LIN {X 0,Y 426.139,Z 463.604,A -85,B 0,C 180,E1 -9930.748,E2 -9930.748} C_VEL
LIN {X 0,Y 426.519,Z 456.049,A -85,B 0,C 180,E1 -9931.425,E2 -9931.425} C_VEL
LIN {X 0,Y 426.812,Z 447.127,A -85,B 0,C 180,E1 -9932.076,E2 -9932.076} C_VEL
LIN {X 0,Y 427.163,Z 437.86,A -85,B 0,C 180,E1 -9932.604,E2 -9932.604} C_VEL
LIN {X 0,Y 427.406,Z 427.667,A -85,B 0,C 180,E1 -9933.038,E2 -9933.038} C_VEL
LIN {X 0,Y 427.627,Z 415.432,A -85,B 0,C 180,E1 -9933.376,E2 -9933.376} C_VEL
LIN {X 0,Y 428.378,Z 356.063,A -85,B 0,C 180,E1 -9934.529,E2 -9934.529} C_VEL
LIN {X 0,Y 425.875,Z 339.164,A -85,B 0,C 180,E1 -9934.972,E2 -9934.972} C_VEL
LIN {X 0,Y 426.543,Z 323.121,A -85,B 0,C 180,E1 -9938.192,E2 -9938.192} C_VEL
LIN {X 0,Y 427.303,Z 307.169,A -85,B 0,C 180,E1 -9941.454,E2 -9941.454} C_VEL
LIN {X 0,Y 427.541,Z 299.568,A -85,B 0,C 180,E1 -9943.038,E2 -9943.038} C_VEL
LIN {X 0,Y 425.324,Z 287.505,A -85,B 0,C 180,E1 -9945.749,E2 -9945.749} C_VEL
LIN {X 0,Y 425.264,Z 287.509,A -85,B 0,C 180,E1 -9948.623,E2 -9948.623} C_VEL
LIN {X 0,Y 425.272,Z 287.509,A -85,B 0,C 180,E1 -9951.101,E2 -9951.101} C_VEL
LIN {X 0,Y 425.29,Z 287.504,A -85,B 0,C 180,E1 -9954.665,E2 -9954.665} C_VEL
LIN {X 0,Y 425.26,Z 287.513,A -85,B 0,C 180,E1 -9958.074,E2 -9958.074} C_VEL
LIN {X 0,Y 425.296,Z 287.504,A -85,B 0,C 180,E1 -9961.366,E2 -9961.366} C_VEL
LIN {X 0,Y 425.26,Z 287.512,A -85,B 0,C 180,E1 -9964.553,E2 -9964.553} C_VEL
LIN {X 0,Y 425.293,Z 287.504,A -85,B 0,C 180,E1 -9967.731,E2 -9967.731} C_VEL
LIN {X 0,Y 425.333,Z 287.501,A -85,B 0,C 180,E1 -9971.096,E2 -9971.096} C_VEL
LIN {X 0,Y 424.637,Z 287.586,A -85,B 0,C 180,E1 -9971.886,E2 -9971.886} C_VEL
LIN {X 0,Y 421.762,Z 287.946,A -85,B 0,C 180,E1 -9973.17,E2 -9973.17} C_VEL
LIN {X 0,Y 419.363,Z 288.243,A -85,B 0,C 180,E1 -9974.207,E2 -9974.207} C_VEL
LIN {X 0,Y 418.359,Z 288.374,A -85,B 0,C 180,E1 -9975.008,E2 -9975.008} C_VEL
LIN {X 0,Y 418.29,Z 288.377,A -85,B 0,C 180,E1 -9975.279,E2 -9975.279} C_VEL
LIN {X 0,Y 418.316,Z 288.373,A -85,B 0,C 180,E1 -9978.368,E2 -9978.368} C_VEL
LIN {X 0,Y 418.451,Z 288.355,A -85,B 0,C 180,E1 -9982.277,E2 -9982.277} C_VEL
LIN {X 0,Y 418.474,Z 288.353,A -85,B 0,C 180,E1 -9984.215,E2 -9984.215} C_VEL
LIN {X 0,Y 418.536,Z 288.348,A -85,B 0,C 180,E1 -9988.074,E2 -9988.074} C_VEL
LIN {X 0,Y 418.409,Z 288.361,A -85,B 0,C 180,E1 -9990.96,E2 -9990.96} C_VEL
LIN {X 0,Y 418.47,Z 288.353,A -85,B 0,C 180,E1 -9992.886,E2 -9992.886} C_VEL
LIN {X 0,Y 418.471,Z 288.358,A -85,B 0,C 180,E1 -9995.781,E2 -9995.781} C_VEL
LIN {X 0,Y 418.369,Z 288.368,A -85,B 0,C 180,E1 -9998.693,E2 -9998.693} C_VEL
LIN {X 0,Y 418.31,Z 288.374,A -85,B 0,C 180,E1 -10001.628,E2 -10001.628} C_VEL
LIN {X 0,Y 418.297,Z 288.383,A -85,B 0,C 180,E1 -10004.594,E2 -10004.594} C_VEL
LIN {X 0,Y 418.275,Z 288.378,A -85,B 0,C 180,E1 -10007.6,E2 -10007.6} C_VEL
LIN {X 0,Y 418.243,Z 288.386,A -85,B 0,C 180,E1 -10010.659,E2 -10010.659} C_VEL
LIN {X 0,Y 418.263,Z 288.38,A -85,B 0,C 180,E1 -10013.778,E2 -10013.778} C_VEL
LIN {X 0,Y 418.212,Z 288.39,A -85,B 0,C 180,E1 -10017.043,E2 -10017.043} C_VEL
LIN {X 0,Y 418.227,Z 288.384,A -85,B 0,C 180,E1 -10020.268,E2 -10020.268} C_VEL
LIN {X 0,Y 418.23,Z 288.392,A -85,B 0,C 180,E1 -10023.673,E2 -10023.673} C_VEL
LIN {X 0,Y 418.217,Z 288.386,A -85,B 0,C 180,E1 -10027.22,E2 -10027.22} C_VEL
LIN {X 0,Y 418.219,Z 288.388,A -85,B 0,C 180,E1 -10029.678,E2 -10029.678} C_VEL
LIN {X 0,Y 418.201,Z 288.393,A -85,B 0,C 180,E1 -10032.316,E2 -10032.316} C_VEL
LIN {X 0,Y 418.206,Z 288.386,A -85,B 0,C 180,E1 -10035.104,E2 -10035.104} C_VEL
LIN {X 0,Y 418.208,Z 288.387,A -85,B 0,C 180,E1 -10037.762,E2 -10037.762} C_VEL
LIN {X 0,Y 418.218,Z 288.393,A -85,B 0,C 180,E1 -10040.615,E2 -10040.615} C_VEL
LIN {X 0,Y 418.204,Z 288.386,A -85,B 0,C 180,E1 -10043.971,E2 -10043.971} C_VEL
LIN {X 0,Y 418.201,Z 288.389,A -85,B 0,C 180,E1 -10047.467,E2 -10047.467} C_VEL
LIN {X 0,Y 418.233,Z 288.387,A -85,B 0,C 180,E1 -10050.89,E2 -10050.89} C_VEL
LIN {X 0,Y 418.224,Z 288.385,A -85,B 0,C 180,E1 -10054.092,E2 -10054.092} C_VEL
LIN {X 0,Y 418.185,Z 288.393,A -85,B 0,C 180,E1 -10057.26,E2 -10057.26} C_VEL
LIN {X 0,Y 418.232,Z 288.384,A -85,B 0,C 180,E1 -10060.361,E2 -10060.361} C_VEL
LIN {X 0,Y 418.264,Z 288.381,A -85,B 0,C 180,E1 -10063.402,E2 -10063.402} C_VEL
LIN {X 0,Y 418.302,Z 288.374,A -85,B 0,C 180,E1 -10066.992,E2 -10066.992} C_VEL
LIN {X 0,Y 418.303,Z 288.383,A -85,B 0,C 180,E1 -10070.327,E2 -10070.327} C_VEL
LIN {X 0,Y 418.439,Z 288.358,A -85,B 0,C 180,E1 -10073.248,E2 -10073.248} C_VEL
LIN {X 0,Y 418.29,Z 288.377,A -85,B 0,C 180,E1 -10075.18,E2 -10075.18} C_VEL
LIN {X 0,Y 418.489,Z 288.352,A -85,B 0,C 180,E1 -10078.075,E2 -10078.075} C_VEL
LIN {X 0,Y 418.614,Z 288.335,A -85,B 0,C 180,E1 -10079.999,E2 -10079.999} C_VEL
LIN {X 0,Y 418.46,Z 288.36,A -85,B 0,C 180,E1 -10082.888,E2 -10082.888} C_VEL
LIN {X 0,Y 418.437,Z 288.359,A -85,B 0,C 180,E1 -10086.751,E2 -10086.751} C_VEL
LIN {X 0,Y 418.286,Z 288.381,A -85,B 0,C 180,E1 -10089.672,E2 -10089.672} C_VEL
LIN {X 0,Y 418.301,Z 288.375,A -85,B 0,C 180,E1 -10093.007,E2 -10093.007} C_VEL
LIN {X 0,Y 418.258,Z 288.38,A -85,B 0,C 180,E1 -10096.736,E2 -10096.736} C_VEL
LIN {X 0,Y 418.22,Z 288.39,A -85,B 0,C 180,E1 -10099.792,E2 -10099.792} C_VEL
LIN {X 0,Y 418.189,Z 288.39,A -85,B 0,C 180,E1 -10102.738,E2 -10102.738} C_VEL
LIN {X 0,Y 418.221,Z 288.387,A -85,B 0,C 180,E1 -10105.907,E2 -10105.907} C_VEL
LIN {X 0,Y 418.218,Z 288.386,A -85,B 0,C 180,E1 -10109.165,E2 -10109.165} C_VEL
LIN {X 0,Y 418.212,Z 288.393,A -85,B 0,C 180,E1 -10112.847,E2 -10112.847} C_VEL
LIN {X 0,Y 418.203,Z 288.387,A -85,B 0,C 180,E1 -10116.241,E2 -10116.241} C_VEL
LIN {X 0,Y 418.204,Z 288.388,A -85,B 0,C 180,E1 -10119.687,E2 -10119.687} C_VEL
LIN {X 0,Y 418.186,Z 288.389,A -85,B 0,C 180,E1 -10122.324,E2 -10122.324} C_VEL
LIN {X 0,Y 418.2,Z 288.39,A -85,B 0,C 180,E1 -10125.112,E2 -10125.112} C_VEL
LIN {X 0,Y 418.207,Z 288.393,A -85,B 0,C 180,E1 -10127.771,E2 -10127.771} C_VEL
LIN {X 0,Y 418.207,Z 288.39,A -85,B 0,C 180,E1 -10131.56,E2 -10131.56} C_VEL
LIN {X 0,Y 418.224,Z 288.384,A -85,B 0,C 180,E1 -10135.162,E2 -10135.162} C_VEL
LIN {X 0,Y 418.219,Z 288.385,A -85,B 0,C 180,E1 -10137.476,E2 -10137.476} C_VEL
LIN {X 0,Y 418.239,Z 288.388,A -85,B 0,C 180,E1 -10140.902,E2 -10140.902} C_VEL
LIN {X 0,Y 418.255,Z 288.523,A -85,B 0,C 180,E1 -10142.033,E2 -10142.033} C_VEL
LIN {X 0,Y 421.967,Z 305.233,A -85,B 0,C 180,E1 -10145.136,E2 -10145.136} C_VEL
LIN {X 0,Y 422.416,Z 308.453,A -85,B 0,C 180,E1 -10145.706,E2 -10145.706} C_VEL
LIN {X 0,Y 421.093,Z 327.942,A -85,B 0,C 180,E1 -10148.918,E2 -10148.918} C_VEL
LIN {X 0,Y 420.029,Z 345.035,A -85,B 0,C 180,E1 -10151.662,E2 -10151.662} C_VEL
LIN {X 0,Y 422.513,Z 365.547,A -85,B 0,C 180,E1 -10152.142,E2 -10152.142} C_VEL
LIN {X 0,Y 421.378,Z 450.417,A -85,B 0,C 180,E1 -10153.719,E2 -10153.719} C_VEL
LIN {X 0,Y 421.099,Z 459.636,A -85,B 0,C 180,E1 -10153.988,E2 -10153.988} C_VEL
LIN {X 0,Y 420.726,Z 469.267,A -85,B 0,C 180,E1 -10154.377,E2 -10154.377} C_VEL
LIN {X 0,Y 420.344,Z 478.447,A -85,B 0,C 180,E1 -10154.86,E2 -10154.86} C_VEL
LIN {X 0,Y 419.758,Z 489.136,A -85,B 0,C 180,E1 -10155.582,E2 -10155.582} C_VEL
LIN {X 0,Y 419.287,Z 499.136,A -85,B 0,C 180,E1 -10156.432,E2 -10156.432} C_VEL
LIN {X 0,Y 418.893,Z 506.591,A -85,B 0,C 180,E1 -10157.182,E2 -10157.182} C_VEL
LIN {X 0,Y 418.352,Z 516.259,A -85,B 0,C 180,E1 -10158.373,E2 -10158.373} C_VEL
LIN {X 0,Y 417.931,Z 522.899,A -85,B 0,C 180,E1 -10159.343,E2 -10159.343} C_VEL
LIN {X 0,Y 417.616,Z 529.845,A -85,B 0,C 180,E1 -10160.559,E2 -10160.559} C_VEL
LIN {X 0,Y 417.407,Z 535.619,A -85,B 0,C 180,E1 -10161.775,E2 -10161.775} C_VEL
LIN {X 0,Y 417.222,Z 541.176,A -85,B 0,C 180,E1 -10163.231,E2 -10163.231} C_VEL
LIN {X 0,Y 417.147,Z 545.5,A -85,B 0,C 180,E1 -10164.686,E2 -10164.686} C_VEL
LIN {X 0,Y 417.054,Z 548.703,A -85,B 0,C 180,E1 -10166.137,E2 -10166.137} C_VEL
LIN {X 0,Y 417.152,Z 550.338,A -85,B 0,C 180,E1 -10167.105,E2 -10167.105} C_VEL
LIN {X 0,Y 417.104,Z 552.078,A -85,B 0,C 180,E1 -10169.037,E2 -10169.037} C_VEL
LIN {X 0,Y 417.117,Z 552.372,A -85,B 0,C 180,E1 -10170.002,E2 -10170.002} C_VEL
LIN {X 0,Y 417.118,Z 551.594,A -85,B 0,C 180,E1 -10171.933,E2 -10171.933} C_VEL
LIN {X 0,Y 417.122,Z 550.564,A -85,B 0,C 180,E1 -10172.899,E2 -10172.899} C_VEL
LIN {X 0,Y 417.146,Z 547.23,A -85,B 0,C 180,E1 -10174.834,E2 -10174.834} C_VEL
LIN {X 0,Y 417.139,Z 543.557,A -85,B 0,C 180,E1 -10176.264,E2 -10176.264} C_VEL
LIN {X 0,Y 417.301,Z 538.557,A -85,B 0,C 180,E1 -10177.744,E2 -10177.744} C_VEL
LIN {X 0,Y 417.555,Z 532.315,A -85,B 0,C 180,E1 -10179.202,E2 -10179.202} C_VEL
LIN {X 0,Y 417.871,Z 525.97,A -85,B 0,C 180,E1 -10180.417,E2 -10180.417} C_VEL
LIN {X 0,Y 418.36,Z 518.307,A -85,B 0,C 180,E1 -10181.631,E2 -10181.631} C_VEL
LIN {X 0,Y 418.762,Z 511.042,A -85,B 0,C 180,E1 -10182.603,E2 -10182.603} C_VEL
LIN {X 0,Y 419.366,Z 502.16,A -85,B 0,C 180,E1 -10183.592,E2 -10183.592} C_VEL
LIN {X 0,Y 419.968,Z 493.44,A -85,B 0,C 180,E1 -10184.402,E2 -10184.402} C_VEL
LIN {X 0,Y 420.56,Z 483.816,A -85,B 0,C 180,E1 -10185.136,E2 -10185.136} C_VEL
LIN {X 0,Y 421.18,Z 472.887,A -85,B 0,C 180,E1 -10185.795,E2 -10185.795} C_VEL
LIN {X 0,Y 421.67,Z 462.526,A -85,B 0,C 180,E1 -10186.273,E2 -10186.273} C_VEL
LIN {X 0,Y 422.057,Z 451.679,A -85,B 0,C 180,E1 -10186.631,E2 -10186.631} C_VEL
LIN {X 0,Y 422.44,Z 432.575,A -85,B 0,C 180,E1 -10187.02,E2 -10187.02} C_VEL
LIN {X 0,Y 423.325,Z 363.978,A -85,B 0,C 180,E1 -10188.327,E2 -10188.327} C_VEL
LIN {X 0,Y 420.546,Z 343.811,A -85,B 0,C 180,E1 -10188.906,E2 -10188.906} C_VEL
LIN {X 0,Y 421.697,Z 323.527,A -85,B 0,C 180,E1 -10192.023,E2 -10192.023} C_VEL
LIN {X 0,Y 422.6,Z 308.661,A -85,B 0,C 180,E1 -10194.313,E2 -10194.313} C_VEL
LIN {X 0,Y 421.537,Z 301.939,A -85,B 0,C 180,E1 -10195.465,E2 -10195.465} C_VEL
LIN {X 0,Y 418.732,Z 290.403,A -85,B 0,C 180,E1 -10197.546,E2 -10197.546} C_VEL
LIN {X 0,Y 418.215,Z 288.398,A -85,B 0,C 180,E1 -10197.947,E2 -10197.947} C_VEL
LIN {X 0,Y 418.232,Z 288.393,A -85,B 0,C 180,E1 -10201.019,E2 -10201.019} C_VEL
LIN {X 0,Y 418.24,Z 288.389,A -85,B 0,C 180,E1 -10203.676,E2 -10203.676} C_VEL
LIN {X 0,Y 418.23,Z 288.391,A -85,B 0,C 180,E1 -10207.223,E2 -10207.223} C_VEL
LIN {X 0,Y 418.239,Z 288.391,A -85,B 0,C 180,E1 -10209.681,E2 -10209.681} C_VEL
LIN {X 0,Y 418.219,Z 288.392,A -85,B 0,C 180,E1 -10212.32,E2 -10212.32} C_VEL
LIN {X 0,Y 418.224,Z 288.389,A -85,B 0,C 180,E1 -10215.108,E2 -10215.108} C_VEL
LIN {X 0,Y 418.24,Z 288.387,A -85,B 0,C 180,E1 -10217.767,E2 -10217.767} C_VEL
LIN {X 0,Y 418.249,Z 288.385,A -85,B 0,C 180,E1 -10220.616,E2 -10220.616} C_VEL
LIN {X 0,Y 418.227,Z 288.389,A -85,B 0,C 180,E1 -10223.975,E2 -10223.975} C_VEL
LIN {X 0,Y 418.237,Z 288.377,A -85,B 0,C 180,E1 -10227.155,E2 -10227.155} C_VEL
LIN {X 0,Y 418.254,Z 288.38,A -85,B 0,C 180,E1 -10230.893,E2 -10230.893} C_VEL
LIN {X 0,Y 418.251,Z 288.383,A -85,B 0,C 180,E1 -10234.095,E2 -10234.095} C_VEL
LIN {X 0,Y 418.252,Z 288.384,A -85,B 0,C 180,E1 -10237.536,E2 -10237.536} C_VEL
LIN {X 0,Y 418.291,Z 288.382,A -85,B 0,C 180,E1 -10240.365,E2 -10240.365} C_VEL
LIN {X 0,Y 418.29,Z 288.381,A -85,B 0,C 180,E1 -10243.404,E2 -10243.404} C_VEL
LIN {X 0,Y 418.329,Z 288.378,A -85,B 0,C 180,E1 -10246.994,E2 -10246.994} C_VEL
LIN {X 0,Y 418.317,Z 288.381,A -85,B 0,C 180,E1 -10250.329,E2 -10250.329} C_VEL
LIN {X 0,Y 418.46,Z 288.367,A -85,B 0,C 180,E1 -10253.249,E2 -10253.249} C_VEL
LIN {X 0,Y 418.308,Z 288.384,A -85,B 0,C 180,E1 -10255.182,E2 -10255.182} C_VEL
LIN {X 0,Y 418.298,Z 288.47,A -85,B 0,C 180,E1 -10256.268,E2 -10256.268} C_VEL
LIN {X 0,Y 420.461,Z 296.073,A -85,B 0,C 180,E1 -10257.606,E2 -10257.606} C_VEL
LIN {X 0,Y 420.112,Z 313.168,A -85,B 0,C 180,E1 -10260.24,E2 -10260.24} C_VEL
LIN {X 0,Y 419.618,Z 336.301,A -85,B 0,C 180,E1 -10263.842,E2 -10263.842} C_VEL
LIN {X 0,Y 419.579,Z 337.849,A -85,B 0,C 180,E1 -10264.083,E2 -10264.083} C_VEL
LIN {X 0,Y 422.854,Z 357.107,A -85,B 0,C 180,E1 -10264.708,E2 -10264.708} C_VEL
LIN {X 0,Y 421.622,Z 422.931,A -85,B 0,C 180,E1 -10266.161,E2 -10266.161} C_VEL
LIN {X 0,Y 421.289,Z 434.723,A -85,B 0,C 180,E1 -10266.586,E2 -10266.586} C_VEL
LIN {X 0,Y 420.807,Z 445.935,A -85,B 0,C 180,E1 -10267.196,E2 -10267.196} C_VEL
LIN {X 0,Y 420.457,Z 454.507,A -85,B 0,C 180,E1 -10267.806,E2 -10267.806} C_VEL
LIN {X 0,Y 419.928,Z 462.922,A -85,B 0,C 180,E1 -10268.542,E2 -10268.542} C_VEL
LIN {X 0,Y 419.395,Z 471.07,A -85,B 0,C 180,E1 -10269.418,E2 -10269.418} C_VEL
LIN {X 0,Y 418.952,Z 478.475,A -85,B 0,C 180,E1 -10270.39,E2 -10270.39} C_VEL
LIN {X 0,Y 418.474,Z 486.143,A -85,B 0,C 180,E1 -10271.627,E2 -10271.627} C_VEL
LIN {X 0,Y 418.056,Z 492.045,A -85,B 0,C 180,E1 -10272.843,E2 -10272.843} C_VEL
LIN {X 0,Y 417.718,Z 496.891,A -85,B 0,C 180,E1 -10274.121,E2 -10274.121} C_VEL
LIN {X 0,Y 417.566,Z 499.938,A -85,B 0,C 180,E1 -10275.123,E2 -10275.123} C_VEL
LIN {X 0,Y 417.303,Z 503.22,A -85,B 0,C 180,E1 -10276.637,E2 -10276.637} C_VEL
LIN {X 0,Y 417.153,Z 504.725,A -85,B 0,C 180,E1 -10277.654,E2 -10277.654} C_VEL
LIN {X 0,Y 417.093,Z 505.659,A -85,B 0,C 180,E1 -10278.673,E2 -10278.673} C_VEL
LIN {X 0,Y 417.029,Z 505.956,A -85,B 0,C 180,E1 -10279.698,E2 -10279.698} C_VEL
LIN {X 0,Y 417.023,Z 505.653,A -85,B 0,C 180,E1 -10280.727,E2 -10280.727} C_VEL
LIN {X 0,Y 417.098,Z 504.436,A -85,B 0,C 180,E1 -10282.077,E2 -10282.077} C_VEL
LIN {X 0,Y 417.309,Z 501.253,A -85,B 0,C 180,E1 -10283.841,E2 -10283.841} C_VEL
LIN {X 0,Y 417.419,Z 498.485,A -85,B 0,C 180,E1 -10284.893,E2 -10284.893} C_VEL
LIN {X 0,Y 417.616,Z 493.932,A -85,B 0,C 180,E1 -10286.197,E2 -10286.197} C_VEL
LIN {X 0,Y 417.843,Z 489.187,A -85,B 0,C 180,E1 -10287.28,E2 -10287.28} C_VEL
LIN {X 0,Y 418.158,Z 483.464,A -85,B 0,C 180,E1 -10288.347,E2 -10288.347} C_VEL
LIN {X 0,Y 418.488,Z 476.42,A -85,B 0,C 180,E1 -10289.421,E2 -10289.421} C_VEL
LIN {X 0,Y 418.872,Z 468.901,A -85,B 0,C 180,E1 -10290.362,E2 -10290.362} C_VEL
LIN {X 0,Y 419.355,Z 459.678,A -85,B 0,C 180,E1 -10291.301,E2 -10291.301} C_VEL
LIN {X 0,Y 419.807,Z 448.412,A -85,B 0,C 180,E1 -10292.18,E2 -10292.18} C_VEL
LIN {X 0,Y 420.156,Z 439.421,A -85,B 0,C 180,E1 -10292.718,E2 -10292.718} C_VEL
LIN {X 0,Y 420.447,Z 429.741,A -85,B 0,C 180,E1 -10293.156,E2 -10293.156} C_VEL
LIN {X 0,Y 420.612,Z 420.061,A -85,B 0,C 180,E1 -10293.463,E2 -10293.463} C_VEL
LIN {X 0,Y 421.449,Z 356.576,A -85,B 0,C 180,E1 -10294.752,E2 -10294.752} C_VEL
LIN {X 0,Y 418.878,Z 339.127,A -85,B 0,C 180,E1 -10295.226,E2 -10295.226} C_VEL
LIN {X 0,Y 419.627,Z 322.538,A -85,B 0,C 180,E1 -10298.6,E2 -10298.6} C_VEL
LIN {X 0,Y 420.4,Z 306.335,A -85,B 0,C 180,E1 -10301.967,E2 -10301.967} C_VEL
LIN {X 0,Y 420.532,Z 300.268,A -85,B 0,C 180,E1 -10303.252,E2 -10303.252} C_VEL
LIN {X 0,Y 418.258,Z 288.384,A -85,B 0,C 180,E1 -10305.97,E2 -10305.97} C_VEL
LIN {X 0,Y 418.213,Z 288.392,A -85,B 0,C 180,E1 -10309.133,E2 -10309.133} C_VEL
LIN {X 0,Y 418.23,Z 288.383,A -85,B 0,C 180,E1 -10312.777,E2 -10312.777} C_VEL
LIN {X 0,Y 418.23,Z 288.385,A -85,B 0,C 180,E1 -10316.323,E2 -10316.323} C_VEL
LIN {X 0,Y 418.238,Z 288.387,A -85,B 0,C 180,E1 -10319.728,E2 -10319.728} C_VEL
LIN {X 0,Y 418.21,Z 288.386,A -85,B 0,C 180,E1 -10323.017,E2 -10323.017} C_VEL
LIN {X 0,Y 418.256,Z 288.386,A -85,B 0,C 180,E1 -10326.217,E2 -10326.217} C_VEL
LIN {X 0,Y 418.249,Z 288.381,A -85,B 0,C 180,E1 -10329.337,E2 -10329.337} C_VEL
LIN {X 0,Y 418.282,Z 288.381,A -85,B 0,C 180,E1 -10332.396,E2 -10332.396} C_VEL
LIN {X 0,Y 418.29,Z 288.377,A -85,B 0,C 180,E1 -10335.279,E2 -10335.279} C_VEL
LIN {X 0,Y 417.66,Z 288.46,A -85,B 0,C 180,E1 -10336.083,E2 -10336.083} C_VEL
LIN {X 0,Y 414.822,Z 288.819,A -85,B 0,C 180,E1 -10337.39,E2 -10337.39} C_VEL
LIN {X 0,Y 412.398,Z 289.12,A -85,B 0,C 180,E1 -10338.445,E2 -10338.445} C_VEL
LIN {X 0,Y 411.354,Z 289.246,A -85,B 0,C 180,E1 -10339.26,E2 -10339.26} C_VEL
LIN {X 0,Y 411.269,Z 289.253,A -85,B 0,C 180,E1 -10339.537,E2 -10339.537} C_VEL
LIN {X 0,Y 411.395,Z 289.24,A -85,B 0,C 180,E1 -10343.131,E2 -10343.131} C_VEL
LIN {X 0,Y 411.287,Z 289.252,A -85,B 0,C 180,E1 -10345.097,E2 -10345.097} C_VEL
LIN {X 0,Y 411.505,Z 289.224,A -85,B 0,C 180,E1 -10348.041,E2 -10348.041} C_VEL
LIN {X 0,Y 411.379,Z 289.237,A -85,B 0,C 180,E1 -10350.977,E2 -10350.977} C_VEL
LIN {X 0,Y 411.428,Z 289.23,A -85,B 0,C 180,E1 -10352.935,E2 -10352.935} C_VEL
LIN {X 0,Y 411.392,Z 289.236,A -85,B 0,C 180,E1 -10356.865,E2 -10356.865} C_VEL
LIN {X 0,Y 411.281,Z 289.251,A -85,B 0,C 180,E1 -10359.836,E2 -10359.836} C_VEL
LIN {X 0,Y 411.304,Z 289.247,A -85,B 0,C 180,E1 -10363.1,E2 -10363.1} C_VEL
LIN {X 0,Y 411.254,Z 289.258,A -85,B 0,C 180,E1 -10366.885,E2 -10366.885} C_VEL
LIN {X 0,Y 411.225,Z 289.256,A -85,B 0,C 180,E1 -10369.983,E2 -10369.983} C_VEL
LIN {X 0,Y 411.186,Z 289.268,A -85,B 0,C 180,E1 -10373.144,E2 -10373.144} C_VEL
LIN {X 0,Y 411.175,Z 289.262,A -85,B 0,C 180,E1 -10376.38,E2 -10376.38} C_VEL
LIN {X 0,Y 411.184,Z 289.266,A -85,B 0,C 180,E1 -10379.708,E2 -10379.708} C_VEL
LIN {X 0,Y 411.19,Z 289.262,A -85,B 0,C 180,E1 -10383.151,E2 -10383.151} C_VEL
LIN {X 0,Y 411.172,Z 289.263,A -85,B 0,C 180,E1 -10386.548,E2 -10386.548} C_VEL
LIN {X 0,Y 411.184,Z 289.265,A -85,B 0,C 180,E1 -10389.722,E2 -10389.722} C_VEL
LIN {X 0,Y 411.145,Z 289.266,A -85,B 0,C 180,E1 -10393.129,E2 -10393.129} C_VEL
LIN {X 0,Y 411.138,Z 289.269,A -85,B 0,C 180,E1 -10395.877,E2 -10395.877} C_VEL
LIN {X 0,Y 411.131,Z 289.272,A -85,B 0,C 180,E1 -10398.767,E2 -10398.767} C_VEL
LIN {X 0,Y 411.168,Z 289.263,A -85,B 0,C 180,E1 -10401.827,E2 -10401.827} C_VEL
LIN {X 0,Y 411.164,Z 289.269,A -85,B 0,C 180,E1 -10405.119,E2 -10405.119} C_VEL
LIN {X 0,Y 411.123,Z 289.268,A -85,B 0,C 180,E1 -10407.998,E2 -10407.998} C_VEL
LIN {X 0,Y 411.18,Z 289.268,A -85,B 0,C 180,E1 -10411.406,E2 -10411.406} C_VEL
LIN {X 0,Y 411.193,Z 289.265,A -85,B 0,C 180,E1 -10413.615,E2 -10413.615} C_VEL
LIN {X 0,Y 411.149,Z 289.266,A -85,B 0,C 180,E1 -10416.849,E2 -10416.849} C_VEL
LIN {X 0,Y 411.164,Z 289.268,A -85,B 0,C 180,E1 -10420.049,E2 -10420.049} C_VEL
LIN {X 0,Y 411.213,Z 289.258,A -85,B 0,C 180,E1 -10423.129,E2 -10423.129} C_VEL
LIN {X 0,Y 411.261,Z 289.252,A -85,B 0,C 180,E1 -10426.89,E2 -10426.89} C_VEL
LIN {X 0,Y 411.252,Z 289.258,A -85,B 0,C 180,E1 -10430.16,E2 -10430.16} C_VEL
LIN {X 0,Y 411.406,Z 289.234,A -85,B 0,C 180,E1 -10433.132,E2 -10433.132} C_VEL
LIN {X 0,Y 411.261,Z 289.254,A -85,B 0,C 180,E1 -10435.098,E2 -10435.098} C_VEL
LIN {X 0,Y 411.459,Z 289.227,A -85,B 0,C 180,E1 -10438.042,E2 -10438.042} C_VEL
LIN {X 0,Y 411.584,Z 289.211,A -85,B 0,C 180,E1 -10439.999,E2 -10439.999} C_VEL
LIN {X 0,Y 411.416,Z 289.239,A -85,B 0,C 180,E1 -10442.937,E2 -10442.937} C_VEL
LIN {X 0,Y 411.405,Z 289.236,A -85,B 0,C 180,E1 -10446.867,E2 -10446.867} C_VEL
LIN {X 0,Y 411.239,Z 289.257,A -85,B 0,C 180,E1 -10449.84,E2 -10449.84} C_VEL
LIN {X 0,Y 411.259,Z 289.253,A -85,B 0,C 180,E1 -10453.109,E2 -10453.109} C_VEL
LIN {X 0,Y 411.205,Z 289.258,A -85,B 0,C 180,E1 -10456.89,E2 -10456.89} C_VEL
LIN {X 0,Y 411.18,Z 289.269,A -85,B 0,C 180,E1 -10459.989,E2 -10459.989} C_VEL
LIN {X 0,Y 411.154,Z 289.265,A -85,B 0,C 180,E1 -10463.15,E2 -10463.15} C_VEL
LIN {X 0,Y 411.189,Z 289.269,A -85,B 0,C 180,E1 -10466.384,E2 -10466.384} C_VEL
LIN {X 0,Y 411.154,Z 289.265,A -85,B 0,C 180,E1 -10469.716,E2 -10469.716} C_VEL
LIN {X 0,Y 411.163,Z 289.267,A -85,B 0,C 180,E1 -10473.159,E2 -10473.159} C_VEL
LIN {X 0,Y 411.151,Z 289.268,A -85,B 0,C 180,E1 -10476.556,E2 -10476.556} C_VEL
LIN {X 0,Y 411.169,Z 289.264,A -85,B 0,C 180,E1 -10479.73,E2 -10479.73} C_VEL
LIN {X 0,Y 411.134,Z 289.272,A -85,B 0,C 180,E1 -10483.138,E2 -10483.138} C_VEL
LIN {X 0,Y 411.133,Z 289.271,A -85,B 0,C 180,E1 -10485.885,E2 -10485.885} C_VEL
LIN {X 0,Y 411.13,Z 289.268,A -85,B 0,C 180,E1 -10488.776,E2 -10488.776} C_VEL
LIN {X 0,Y 411.154,Z 289.271,A -85,B 0,C 180,E1 -10492.029,E2 -10492.029} C_VEL
LIN {X 0,Y 411.176,Z 289.262,A -85,B 0,C 180,E1 -10495.128,E2 -10495.128} C_VEL
LIN {X 0,Y 411.14,Z 289.272,A -85,B 0,C 180,E1 -10498.006,E2 -10498.006} C_VEL
LIN {X 0,Y 411.199,Z 289.265,A -85,B 0,C 180,E1 -10501.693,E2 -10501.693} C_VEL
LIN {X 0,Y 414.962,Z 306.311,A -85,B 0,C 180,E1 -10504.955,E2 -10504.955} C_VEL
LIN {X 0,Y 415.512,Z 309.742,A -85,B 0,C 180,E1 -10505.577,E2 -10505.577} C_VEL
LIN {X 0,Y 414.024,Z 330.205,A -85,B 0,C 180,E1 -10509.005,E2 -10509.005} C_VEL
LIN {X 0,Y 413.051,Z 344.849,A -85,B 0,C 180,E1 -10511.412,E2 -10511.412} C_VEL
LIN {X 0,Y 415.654,Z 367.115,A -85,B 0,C 180,E1 -10511.939,E2 -10511.939} C_VEL
LIN {X 0,Y 414.469,Z 449.48,A -85,B 0,C 180,E1 -10513.503,E2 -10513.503} C_VEL
LIN {X 0,Y 414.14,Z 458.907,A -85,B 0,C 180,E1 -10513.775,E2 -10513.775} C_VEL
LIN {X 0,Y 413.765,Z 468.654,A -85,B 0,C 180,E1 -10514.171,E2 -10514.171} C_VEL
LIN {X 0,Y 413.321,Z 478.84,A -85,B 0,C 180,E1 -10514.722,E2 -10514.722} C_VEL
LIN {X 0,Y 412.737,Z 489.395,A -85,B 0,C 180,E1 -10515.457,E2 -10515.457} C_VEL
LIN {X 0,Y 412.349,Z 498.056,A -85,B 0,C 180,E1 -10516.199,E2 -10516.199} C_VEL
LIN {X 0,Y 411.771,Z 507.515,A -85,B 0,C 180,E1 -10517.184,E2 -10517.184} C_VEL
LIN {X 0,Y 411.335,Z 515.42,A -85,B 0,C 180,E1 -10518.172,E2 -10518.172} C_VEL
LIN {X 0,Y 410.909,Z 522.149,A -85,B 0,C 180,E1 -10519.159,E2 -10519.159} C_VEL
LIN {X 0,Y 410.555,Z 529.168,A -85,B 0,C 180,E1 -10520.395,E2 -10520.395} C_VEL
LIN {X 0,Y 410.33,Z 535.005,A -85,B 0,C 180,E1 -10521.632,E2 -10521.632} C_VEL
LIN {X 0,Y 410.154,Z 540.617,A -85,B 0,C 180,E1 -10523.114,E2 -10523.114} C_VEL
LIN {X 0,Y 410.06,Z 544.984,A -85,B 0,C 180,E1 -10524.594,E2 -10524.594} C_VEL
LIN {X 0,Y 409.971,Z 548.225,A -85,B 0,C 180,E1 -10526.07,E2 -10526.07} C_VEL
LIN {X 0,Y 410.066,Z 549.865,A -85,B 0,C 180,E1 -10527.055,E2 -10527.055} C_VEL
LIN {X 0,Y 410.024,Z 551.661,A -85,B 0,C 180,E1 -10529.02,E2 -10529.02} C_VEL
LIN {X 0,Y 410.033,Z 551.953,A -85,B 0,C 180,E1 -10530.002,E2 -10530.002} C_VEL
LIN {X 0,Y 410.045,Z 551.228,A -85,B 0,C 180,E1 -10531.966,E2 -10531.966} C_VEL
LIN {X 0,Y 410.02,Z 550.193,A -85,B 0,C 180,E1 -10532.949,E2 -10532.949} C_VEL
LIN {X 0,Y 410.052,Z 546.902,A -85,B 0,C 180,E1 -10534.918,E2 -10534.918} C_VEL
LIN {X 0,Y 410.066,Z 543.167,A -85,B 0,C 180,E1 -10536.397,E2 -10536.397} C_VEL
LIN {X 0,Y 410.223,Z 538.259,A -85,B 0,C 180,E1 -10537.879,E2 -10537.879} C_VEL
LIN {X 0,Y 410.516,Z 532.031,A -85,B 0,C 180,E1 -10539.361,E2 -10539.361} C_VEL
LIN {X 0,Y 410.854,Z 525.696,A -85,B 0,C 180,E1 -10540.597,E2 -10540.597} C_VEL
LIN {X 0,Y 411.39,Z 518.044,A -85,B 0,C 180,E1 -10541.83,E2 -10541.83} C_VEL
LIN {X 0,Y 411.817,Z 510.828,A -85,B 0,C 180,E1 -10542.819,E2 -10542.819} C_VEL
LIN {X 0,Y 412.439,Z 502.234,A -85,B 0,C 180,E1 -10543.802,E2 -10543.802} C_VEL
LIN {X 0,Y 413.106,Z 493.215,A -85,B 0,C 180,E1 -10544.659,E2 -10544.659} C_VEL
LIN {X 0,Y 413.713,Z 483.851,A -85,B 0,C 180,E1 -10545.393,E2 -10545.393} C_VEL
LIN {X 0,Y 414.37,Z 473.024,A -85,B 0,C 180,E1 -10546.062,E2 -10546.062} C_VEL
LIN {X 0,Y 414.905,Z 462.014,A -85,B 0,C 180,E1 -10546.578,E2 -10546.578} C_VEL
LIN {X 0,Y 415.251,Z 452.324,A -85,B 0,C 180,E1 -10546.912,E2 -10546.912} C_VEL
LIN {X 0,Y 415.697,Z 433.55,A -85,B 0,C 180,E1 -10547.305,E2 -10547.305} C_VEL
LIN {X 0,Y 416.66,Z 364.602,A -85,B 0,C 180,E1 -10548.648,E2 -10548.648} C_VEL
LIN {X 0,Y 413.754,Z 343.881,A -85,B 0,C 180,E1 -10549.249,E2 -10549.249} C_VEL
LIN {X 0,Y 415.048,Z 322.035,A -85,B 0,C 180,E1 -10552.657,E2 -10552.657} C_VEL
LIN {X 0,Y 415.758,Z 308.95,A -85,B 0,C 180,E1 -10554.731,E2 -10554.731} C_VEL
LIN {X 0,Y 413.326,Z 297.518,A -85,B 0,C 180,E1 -10556.781,E2 -10556.781} C_VEL
LIN {X 0,Y 411.193,Z 289.273,A -85,B 0,C 180,E1 -10558.382,E2 -10558.382} C_VEL
LIN {X 0,Y 411.158,Z 289.272,A -85,B 0,C 180,E1 -10561.997,E2 -10561.997} C_VEL
LIN {X 0,Y 411.202,Z 289.265,A -85,B 0,C 180,E1 -10564.877,E2 -10564.877} C_VEL
LIN {X 0,Y 411.194,Z 289.267,A -85,B 0,C 180,E1 -10568.167,E2 -10568.167} C_VEL
LIN {X 0,Y 411.153,Z 289.274,A -85,B 0,C 180,E1 -10571.227,E2 -10571.227} C_VEL
LIN {X 0,Y 411.165,Z 289.269,A -85,B 0,C 180,E1 -10574.489,E2 -10574.489} C_VEL
LIN {X 0,Y 411.183,Z 289.267,A -85,B 0,C 180,E1 -10578.196,E2 -10578.196} C_VEL
LIN {X 0,Y 411.212,Z 289.261,A -85,B 0,C 180,E1 -10580.776,E2 -10580.776} C_VEL
LIN {X 0,Y 411.181,Z 289.261,A -85,B 0,C 180,E1 -10584.47,E2 -10584.47} C_VEL
LIN {X 0,Y 411.188,Z 289.256,A -85,B 0,C 180,E1 -10586.872,E2 -10586.872} C_VEL
LIN {X 0,Y 411.219,Z 289.259,A -85,B 0,C 180,E1 -10590.642,E2 -10590.642} C_VEL
LIN {X 0,Y 411.217,Z 289.258,A -85,B 0,C 180,E1 -10593.618,E2 -10593.618} C_VEL
LIN {X 0,Y 411.187,Z 289.266,A -85,B 0,C 180,E1 -10596.852,E2 -10596.852} C_VEL
LIN {X 0,Y 411.241,Z 289.259,A -85,B 0,C 180,E1 -10600.031,E2 -10600.031} C_VEL
LIN {X 0,Y 411.238,Z 289.261,A -85,B 0,C 180,E1 -10603.131,E2 -10603.131} C_VEL
LIN {X 0,Y 411.287,Z 289.256,A -85,B 0,C 180,E1 -10606.891,E2 -10606.891} C_VEL
LIN {X 0,Y 411.27,Z 289.258,A -85,B 0,C 180,E1 -10610.161,E2 -10610.161} C_VEL
LIN {X 0,Y 411.425,Z 289.244,A -85,B 0,C 180,E1 -10613.133,E2 -10613.133} C_VEL
LIN {X 0,Y 411.231,Z 289.264,A -85,B 0,C 180,E1 -10615.835,E2 -10615.835} C_VEL
LIN {X 0,Y 413.573,Z 297.373,A -85,B 0,C 180,E1 -10617.322,E2 -10617.322} C_VEL
LIN {X 0,Y 413.691,Z 303.478,A -85,B 0,C 180,E1 -10618.297,E2 -10618.297} C_VEL
LIN {X 0,Y 413.01,Z 325.266,A -85,B 0,C 180,E1 -10621.707,E2 -10621.707} C_VEL
LIN {X 0,Y 412.793,Z 338.159,A -85,B 0,C 180,E1 -10623.722,E2 -10623.722} C_VEL
LIN {X 0,Y 416.168,Z 357.741,A -85,B 0,C 180,E1 -10624.381,E2 -10624.381} C_VEL
LIN {X 0,Y 414.88,Z 423.19,A -85,B 0,C 180,E1 -10625.865,E2 -10625.865} C_VEL
LIN {X 0,Y 414.517,Z 434.284,A -85,B 0,C 180,E1 -10626.267,E2 -10626.267} C_VEL
LIN {X 0,Y 414.097,Z 444.82,A -85,B 0,C 180,E1 -10626.824,E2 -10626.824} C_VEL
LIN {X 0,Y 413.616,Z 455.178,A -85,B 0,C 180,E1 -10627.567,E2 -10627.567} C_VEL
LIN {X 0,Y 413.068,Z 463.539,A -85,B 0,C 180,E1 -10628.316,E2 -10628.316} C_VEL
LIN {X 0,Y 412.561,Z 470.993,A -85,B 0,C 180,E1 -10629.128,E2 -10629.128} C_VEL
LIN {X 0,Y 412.096,Z 478.124,A -85,B 0,C 180,E1 -10630.068,E2 -10630.068} C_VEL
LIN {X 0,Y 411.637,Z 484.456,A -85,B 0,C 180,E1 -10631.074,E2 -10631.074} C_VEL
LIN {X 0,Y 411.148,Z 490.944,A -85,B 0,C 180,E1 -10632.338,E2 -10632.338} C_VEL
LIN {X 0,Y 410.723,Z 496.939,A -85,B 0,C 180,E1 -10633.861,E2 -10633.861} C_VEL
LIN {X 0,Y 410.528,Z 500.064,A -85,B 0,C 180,E1 -10634.88,E2 -10634.88} C_VEL
LIN {X 0,Y 410.267,Z 503.435,A -85,B 0,C 180,E1 -10636.416,E2 -10636.416} C_VEL
LIN {X 0,Y 410.038,Z 505.518,A -85,B 0,C 180,E1 -10637.971,E2 -10637.971} C_VEL
LIN {X 0,Y 409.975,Z 506.318,A -85,B 0,C 180,E1 -10639.476,E2 -10639.476} C_VEL
LIN {X 0,Y 409.947,Z 505.858,A -85,B 0,C 180,E1 -10641.102,E2 -10641.102} C_VEL
LIN {X 0,Y 410.04,Z 504.619,A -85,B 0,C 180,E1 -10642.258,E2 -10642.258} C_VEL
LIN {X 0,Y 410.209,Z 501.935,A -85,B 0,C 180,E1 -10643.743,E2 -10643.743} C_VEL
LIN {X 0,Y 410.322,Z 499.249,A -85,B 0,C 180,E1 -10644.807,E2 -10644.807} C_VEL
LIN {X 0,Y 410.52,Z 494.706,A -85,B 0,C 180,E1 -10646.158,E2 -10646.158} C_VEL
LIN {X 0,Y 410.828,Z 488.8,A -85,B 0,C 180,E1 -10647.51,E2 -10647.51} C_VEL
LIN {X 0,Y 411.134,Z 482.899,A -85,B 0,C 180,E1 -10648.597,E2 -10648.597} C_VEL
LIN {X 0,Y 411.451,Z 477.011,A -85,B 0,C 180,E1 -10649.5,E2 -10649.5} C_VEL
LIN {X 0,Y 411.814,Z 470.262,A -85,B 0,C 180,E1 -10650.37,E2 -10650.37} C_VEL
LIN {X 0,Y 412.224,Z 461.839,A -85,B 0,C 180,E1 -10651.268,E2 -10651.268} C_VEL
LIN {X 0,Y 412.725,Z 451.506,A -85,B 0,C 180,E1 -10652.15,E2 -10652.15} C_VEL
LIN {X 0,Y 413.163,Z 440.777,A -85,B 0,C 180,E1 -10652.834,E2 -10652.834} C_VEL
LIN {X 0,Y 413.452,Z 430.374,A -85,B 0,C 180,E1 -10653.323,E2 -10653.323} C_VEL
LIN {X 0,Y 413.651,Z 420.453,A -85,B 0,C 180,E1 -10653.647,E2 -10653.647} C_VEL
LIN {X 0,Y 414.617,Z 357.744,A -85,B 0,C 180,E1 -10654.955,E2 -10654.955} C_VEL
LIN {X 0,Y 411.878,Z 339.185,A -85,B 0,C 180,E1 -10655.462,E2 -10655.462} C_VEL
LIN {X 0,Y 412.64,Z 323.562,A -85,B 0,C 180,E1 -10658.686,E2 -10658.686} C_VEL
LIN {X 0,Y 413.473,Z 306.976,A -85,B 0,C 180,E1 -10662.175,E2 -10662.175} C_VEL
LIN {X 0,Y 413.541,Z 301.272,A -85,B 0,C 180,E1 -10663.408,E2 -10663.408} C_VEL
LIN {X 0,Y 411.197,Z 289.263,A -85,B 0,C 180,E1 -10666.192,E2 -10666.192} C_VEL
LIN {X 0,Y 411.163,Z 289.272,A -85,B 0,C 180,E1 -10669.496,E2 -10669.496} C_VEL
LIN {X 0,Y 411.178,Z 289.264,A -85,B 0,C 180,E1 -10672.026,E2 -10672.026} C_VEL
LIN {X 0,Y 411.199,Z 289.26,A -85,B 0,C 180,E1 -10675.125,E2 -10675.125} C_VEL
LIN {X 0,Y 411.162,Z 289.271,A -85,B 0,C 180,E1 -10678.004,E2 -10678.004} C_VEL
LIN {X 0,Y 411.172,Z 289.263,A -85,B 0,C 180,E1 -10681.407,E2 -10681.407} C_VEL
LIN {X 0,Y 411.19,Z 289.261,A -85,B 0,C 180,E1 -10684.942,E2 -10684.942} C_VEL
LIN {X 0,Y 411.203,Z 289.26,A -85,B 0,C 180,E1 -10687.914,E2 -10687.914} C_VEL
LIN {X 0,Y 411.221,Z 289.259,A -85,B 0,C 180,E1 -10691.051,E2 -10691.051} C_VEL
LIN {X 0,Y 411.251,Z 289.253,A -85,B 0,C 180,E1 -10694.131,E2 -10694.131} C_VEL
LIN {X 0,Y 411.308,Z 289.251,A -85,B 0,C 180,E1 -10697.165,E2 -10697.165} C_VEL
LIN {X 0,Y 411.269,Z 289.253,A -85,B 0,C 180,E1 -10699.537,E2 -10699.537} C_VEL
LIN {X 0,Y 410.605,Z 289.334,A -85,B 0,C 180,E1 -10700.355,E2 -10700.355} C_VEL
LIN {X 0,Y 407.775,Z 289.688,A -85,B 0,C 180,E1 -10701.686,E2 -10701.686} C_VEL
LIN {X 0,Y 405.406,Z 289.982,A -85,B 0,C 180,E1 -10702.761,E2 -10702.761} C_VEL
LIN {X 0,Y 404.423,Z 290.108,A -85,B 0,C 180,E1 -10703.591,E2 -10703.591} C_VEL
LIN {X 0,Y 404.36,Z 290.112,A -85,B 0,C 180,E1 -10703.872,E2 -10703.872} C_VEL
LIN {X 0,Y 404.473,Z 290.1,A -85,B 0,C 180,E1 -10708.007,E2 -10708.007} C_VEL
LIN {X 0,Y 404.35,Z 290.113,A -85,B 0,C 180,E1 -10710.994,E2 -10710.994} C_VEL
LIN {X 0,Y 404.362,Z 290.111,A -85,B 0,C 180,E1 -10712.987,E2 -10712.987} C_VEL
LIN {X 0,Y 404.368,Z 290.117,A -85,B 0,C 180,E1 -10715.983,E2 -10715.983} C_VEL
LIN {X 0,Y 404.258,Z 290.124,A -85,B 0,C 180,E1 -10718.999,E2 -10718.999} C_VEL
LIN {X 0,Y 404.253,Z 290.128,A -85,B 0,C 180,E1 -10722.038,E2 -10722.038} C_VEL
LIN {X 0,Y 404.201,Z 290.133,A -85,B 0,C 180,E1 -10725.115,E2 -10725.115} C_VEL
LIN {X 0,Y 404.2,Z 290.133,A -85,B 0,C 180,E1 -10728.235,E2 -10728.235} C_VEL
LIN {X 0,Y 404.131,Z 290.142,A -85,B 0,C 180,E1 -10731.415,E2 -10731.415} C_VEL
LIN {X 0,Y 404.145,Z 290.14,A -85,B 0,C 180,E1 -10734.663,E2 -10734.663} C_VEL
LIN {X 0,Y 404.109,Z 290.143,A -85,B 0,C 180,E1 -10738.001,E2 -10738.001} C_VEL
LIN {X 0,Y 404.13,Z 290.14,A -85,B 0,C 180,E1 -10740.281,E2 -10740.281} C_VEL
LIN {X 0,Y 404.127,Z 290.146,A -85,B 0,C 180,E1 -10743.808,E2 -10743.808} C_VEL
LIN {X 0,Y 404.114,Z 290.142,A -85,B 0,C 180,E1 -10746.87,E2 -10746.87} C_VEL
LIN {X 0,Y 404.125,Z 290.148,A -85,B 0,C 180,E1 -10750.075,E2 -10750.075} C_VEL
LIN {X 0,Y 404.125,Z 290.14,A -85,B 0,C 180,E1 -10753.079,E2 -10753.079} C_VEL
LIN {X 0,Y 404.119,Z 290.144,A -85,B 0,C 180,E1 -10755.921,E2 -10755.921} C_VEL
LIN {X 0,Y 404.086,Z 290.152,A -85,B 0,C 180,E1 -10758.63,E2 -10758.63} C_VEL
LIN {X 0,Y 404.118,Z 290.141,A -85,B 0,C 180,E1 -10761.488,E2 -10761.488} C_VEL
LIN {X 0,Y 404.136,Z 290.146,A -85,B 0,C 180,E1 -10764.978,E2 -10764.978} C_VEL
LIN {X 0,Y 404.099,Z 290.145,A -85,B 0,C 180,E1 -10768.438,E2 -10768.438} C_VEL
LIN {X 0,Y 404.155,Z 290.137,A -85,B 0,C 180,E1 -10771.997,E2 -10771.997} C_VEL
LIN {X 0,Y 404.129,Z 290.146,A -85,B 0,C 180,E1 -10775.331,E2 -10775.331} C_VEL
LIN {X 0,Y 404.089,Z 290.145,A -85,B 0,C 180,E1 -10778.577,E2 -10778.577} C_VEL
LIN {X 0,Y 404.158,Z 290.143,A -85,B 0,C 180,E1 -10781.759,E2 -10781.759} C_VEL
LIN {X 0,Y 404.155,Z 290.137,A -85,B 0,C 180,E1 -10784.88,E2 -10784.88} C_VEL
LIN {X 0,Y 404.216,Z 290.134,A -85,B 0,C 180,E1 -10787.957,E2 -10787.957} C_VEL
LIN {X 0,Y 404.353,Z 290.116,A -85,B 0,C 180,E1 -10792.126,E2 -10792.126} C_VEL
LIN {X 0,Y 404.37,Z 290.112,A -85,B 0,C 180,E1 -10794.014,E2 -10794.014} C_VEL
LIN {X 0,Y 404.428,Z 290.103,A -85,B 0,C 180,E1 -10798.008,E2 -10798.008} C_VEL
LIN {X 0,Y 404.554,Z 290.087,A -85,B 0,C 180,E1 -10799.999,E2 -10799.999} C_VEL
LIN {X 0,Y 404.373,Z 290.117,A -85,B 0,C 180,E1 -10802.988,E2 -10802.988} C_VEL
LIN {X 0,Y 404.351,Z 290.116,A -85,B 0,C 180,E1 -10806.988,E2 -10806.988} C_VEL
LIN {X 0,Y 404.206,Z 290.132,A -85,B 0,C 180,E1 -10810.012,E2 -10810.012} C_VEL
LIN {X 0,Y 404.214,Z 290.132,A -85,B 0,C 180,E1 -10813.213,E2 -10813.213} C_VEL
LIN {X 0,Y 404.164,Z 290.135,A -85,B 0,C 180,E1 -10817.008,E2 -10817.008} C_VEL
LIN {X 0,Y 404.115,Z 290.146,A -85,B 0,C 180,E1 -10820.354,E2 -10820.354} C_VEL
LIN {X 0,Y 404.121,Z 290.142,A -85,B 0,C 180,E1 -10823.577,E2 -10823.577} C_VEL
LIN {X 0,Y 404.136,Z 290.14,A -85,B 0,C 180,E1 -10825.769,E2 -10825.769} C_VEL
LIN {X 0,Y 404.148,Z 290.139,A -85,B 0,C 180,E1 -10828.003,E2 -10828.003} C_VEL
LIN {X 0,Y 404.093,Z 290.144,A -85,B 0,C 180,E1 -10831.56,E2 -10831.56} C_VEL
LIN {X 0,Y 404.142,Z 290.145,A -85,B 0,C 180,E1 -10835.02,E2 -10835.02} C_VEL
LIN {X 0,Y 404.111,Z 290.146,A -85,B 0,C 180,E1 -10838.761,E2 -10838.761} C_VEL
LIN {X 0,Y 404.081,Z 290.15,A -85,B 0,C 180,E1 -10841.603,E2 -10841.603} C_VEL
LIN {X 0,Y 404.109,Z 290.142,A -85,B 0,C 180,E1 -10844.526,E2 -10844.526} C_VEL
LIN {X 0,Y 404.103,Z 290.147,A -85,B 0,C 180,E1 -10847.299,E2 -10847.299} C_VEL
LIN {X 0,Y 404.103,Z 290.148,A -85,B 0,C 180,E1 -10849.955,E2 -10849.955} C_VEL
LIN {X 0,Y 404.104,Z 290.143,A -85,B 0,C 180,E1 -10853.13,E2 -10853.13} C_VEL
LIN {X 0,Y 404.113,Z 290.149,A -85,B 0,C 180,E1 -10856.191,E2 -10856.191} C_VEL
LIN {X 0,Y 404.121,Z 290.144,A -85,B 0,C 180,E1 -10859.719,E2 -10859.719} C_VEL
LIN {X 0,Y 404.149,Z 290.251,A -85,B 0,C 180,E1 -10861.472,E2 -10861.472} C_VEL
LIN {X 0,Y 407.928,Z 307.355,A -85,B 0,C 180,E1 -10864.765,E2 -10864.765} C_VEL
LIN {X 0,Y 408.541,Z 312.023,A -85,B 0,C 180,E1 -10865.62,E2 -10865.62} C_VEL
LIN {X 0,Y 406.912,Z 333.565,A -85,B 0,C 180,E1 -10869.285,E2 -10869.285} C_VEL
LIN {X 0,Y 406.098,Z 344.662,A -85,B 0,C 180,E1 -10871.155,E2 -10871.155} C_VEL
LIN {X 0,Y 408.761,Z 367.463,A -85,B 0,C 180,E1 -10871.711,E2 -10871.711} C_VEL
LIN {X 0,Y 407.528,Z 449.794,A -85,B 0,C 180,E1 -10873.311,E2 -10873.311} C_VEL
LIN {X 0,Y 407.189,Z 459.013,A -85,B 0,C 180,E1 -10873.587,E2 -10873.587} C_VEL
LIN {X 0,Y 406.771,Z 469.252,A -85,B 0,C 180,E1 -10874.02,E2 -10874.02} C_VEL
LIN {X 0,Y 406.302,Z 479.234,A -85,B 0,C 180,E1 -10874.58,E2 -10874.58} C_VEL
LIN {X 0,Y 405.718,Z 489.653,A -85,B 0,C 180,E1 -10875.328,E2 -10875.328} C_VEL
LIN {X 0,Y 405.289,Z 498.409,A -85,B 0,C 180,E1 -10876.102,E2 -10876.102} C_VEL
LIN {X 0,Y 404.735,Z 507.593,A -85,B 0,C 180,E1 -10877.085,E2 -10877.085} C_VEL
LIN {X 0,Y 404.311,Z 514.563,A -85,B 0,C 180,E1 -10877.963,E2 -10877.963} C_VEL
LIN {X 0,Y 403.782,Z 522.821,A -85,B 0,C 180,E1 -10879.219,E2 -10879.219} C_VEL
LIN {X 0,Y 403.455,Z 529.666,A -85,B 0,C 180,E1 -10880.478,E2 -10880.478} C_VEL
LIN {X 0,Y 403.267,Z 534.366,A -85,B 0,C 180,E1 -10881.484,E2 -10881.484} C_VEL
LIN {X 0,Y 403.065,Z 540.036,A -85,B 0,C 180,E1 -10882.992,E2 -10882.992} C_VEL
LIN {X 0,Y 402.956,Z 544.452,A -85,B 0,C 180,E1 -10884.498,E2 -10884.498} C_VEL
LIN {X 0,Y 402.892,Z 547.737,A -85,B 0,C 180,E1 -10886.001,E2 -10886.001} C_VEL
LIN {X 0,Y 402.966,Z 549.376,A -85,B 0,C 180,E1 -10887.003,E2 -10887.003} C_VEL
LIN {X 0,Y 402.946,Z 551.243,A -85,B 0,C 180,E1 -10889.003,E2 -10889.003} C_VEL
LIN {X 0,Y 402.952,Z 551.532,A -85,B 0,C 180,E1 -10890.002,E2 -10890.002} C_VEL
LIN {X 0,Y 402.972,Z 550.863,A -85,B 0,C 180,E1 -10892.001,E2 -10892.001} C_VEL
LIN {X 0,Y 402.919,Z 549.821,A -85,B 0,C 180,E1 -10893.001,E2 -10893.001} C_VEL
LIN {X 0,Y 402.959,Z 546.571,A -85,B 0,C 180,E1 -10895.004,E2 -10895.004} C_VEL
LIN {X 0,Y 403,Z 543.004,A -85,B 0,C 180,E1 -10896.46,E2 -10896.46} C_VEL
LIN {X 0,Y 403.165,Z 537.964,A -85,B 0,C 180,E1 -10898.018,E2 -10898.018} C_VEL
LIN {X 0,Y 403.461,Z 531.77,A -85,B 0,C 180,E1 -10899.526,E2 -10899.526} C_VEL
LIN {X 0,Y 403.849,Z 525.482,A -85,B 0,C 180,E1 -10900.783,E2 -10900.783} C_VEL
LIN {X 0,Y 404.429,Z 517.887,A -85,B 0,C 180,E1 -10902.037,E2 -10902.037} C_VEL
LIN {X 0,Y 404.878,Z 510.703,A -85,B 0,C 180,E1 -10903.042,E2 -10903.042} C_VEL
LIN {X 0,Y 405.53,Z 502.149,A -85,B 0,C 180,E1 -10904.042,E2 -10904.042} C_VEL
LIN {X 0,Y 406.329,Z 491.674,A -85,B 0,C 180,E1 -10905.038,E2 -10905.038} C_VEL
LIN {X 0,Y 406.982,Z 482.016,A -85,B 0,C 180,E1 -10905.783,E2 -10905.783} C_VEL
LIN {X 0,Y 407.633,Z 471.961,A -85,B 0,C 180,E1 -10906.399,E2 -10906.399} C_VEL
LIN {X 0,Y 408.168,Z 461.506,A -85,B 0,C 180,E1 -10906.892,E2 -10906.892} C_VEL
LIN {X 0,Y 408.557,Z 451.721,A -85,B 0,C 180,E1 -10907.23,E2 -10907.23} C_VEL
LIN {X 0,Y 409.057,Z 429.911,A -85,B 0,C 180,E1 -10907.692,E2 -10907.692} C_VEL
LIN {X 0,Y 410.042,Z 365.326,A -85,B 0,C 180,E1 -10908.99,E2 -10908.99} C_VEL
LIN {X 0,Y 406.966,Z 343.755,A -85,B 0,C 180,E1 -10909.645,E2 -10909.645} C_VEL
LIN {X 0,Y 408.361,Z 322.343,A -85,B 0,C 180,E1 -10913.05,E2 -10913.05} C_VEL
LIN {X 0,Y 409.027,Z 310.854,A -85,B 0,C 180,E1 -10914.894,E2 -10914.894} C_VEL
LIN {X 0,Y 406.644,Z 299.666,A -85,B 0,C 180,E1 -10916.957,E2 -10916.957} C_VEL
LIN {X 0,Y 404.161,Z 290.149,A -85,B 0,C 180,E1 -10918.815,E2 -10918.815} C_VEL
LIN {X 0,Y 404.134,Z 290.146,A -85,B 0,C 180,E1 -10922.621,E2 -10922.621} C_VEL
LIN {X 0,Y 404.172,Z 290.141,A -85,B 0,C 180,E1 -10925.189,E2 -10925.189} C_VEL
LIN {X 0,Y 404.144,Z 290.145,A -85,B 0,C 180,E1 -10928.756,E2 -10928.756} C_VEL
LIN {X 0,Y 404.112,Z 290.15,A -85,B 0,C 180,E1 -10931.599,E2 -10931.599} C_VEL
LIN {X 0,Y 404.135,Z 290.145,A -85,B 0,C 180,E1 -10934.521,E2 -10934.521} C_VEL
LIN {X 0,Y 404.13,Z 290.145,A -85,B 0,C 180,E1 -10937.295,E2 -10937.295} C_VEL
LIN {X 0,Y 404.154,Z 290.141,A -85,B 0,C 180,E1 -10939.954,E2 -10939.954} C_VEL
LIN {X 0,Y 404.122,Z 290.141,A -85,B 0,C 180,E1 -10943.123,E2 -10943.123} C_VEL
LIN {X 0,Y 404.126,Z 290.143,A -85,B 0,C 180,E1 -10946.187,E2 -10946.187} C_VEL
LIN {X 0,Y 404.132,Z 290.136,A -85,B 0,C 180,E1 -10949.714,E2 -10949.714} C_VEL
LIN {X 0,Y 404.174,Z 290.135,A -85,B 0,C 180,E1 -10953.122,E2 -10953.122} C_VEL
LIN {X 0,Y 404.151,Z 290.141,A -85,B 0,C 180,E1 -10956.425,E2 -10956.425} C_VEL
LIN {X 0,Y 404.203,Z 290.135,A -85,B 0,C 180,E1 -10959.86,E2 -10959.86} C_VEL
LIN {X 0,Y 404.191,Z 290.138,A -85,B 0,C 180,E1 -10962.993,E2 -10962.993} C_VEL
LIN {X 0,Y 404.258,Z 290.131,A -85,B 0,C 180,E1 -10966.939,E2 -10966.939} C_VEL
LIN {X 0,Y 404.236,Z 290.134,A -85,B 0,C 180,E1 -10969.988,E2 -10969.988} C_VEL
LIN {X 0,Y 404.37,Z 290.122,A -85,B 0,C 180,E1 -10973.013,E2 -10973.013} C_VEL
LIN {X 0,Y 404.237,Z 290.321,A -85,B 0,C 180,E1 -10975.451,E2 -10975.451} C_VEL
LIN {X 0,Y 407.001,Z 300.18,A -85,B 0,C 180,E1 -10977.279,E2 -10977.279} C_VEL
LIN {X 0,Y 406.65,Z 314.134,A -85,B 0,C 180,E1 -10979.505,E2 -10979.505} C_VEL
LIN {X 0,Y 405.986,Z 335.873,A -85,B 0,C 180,E1 -10982.977,E2 -10982.977} C_VEL
LIN {X 0,Y 405.947,Z 338.047,A -85,B 0,C 180,E1 -10983.319,E2 -10983.319} C_VEL
LIN {X 0,Y 409.531,Z 358.384,A -85,B 0,C 180,E1 -10984.029,E2 -10984.029} C_VEL
LIN {X 0,Y 409.416,Z 370.076,A -85,B 0,C 180,E1 -10984.308,E2 -10984.308} C_VEL
LIN {X 0,Y 408.15,Z 423.577,A -85,B 0,C 180,E1 -10985.559,E2 -10985.559} C_VEL
LIN {X 0,Y 407.751,Z 435.289,A -85,B 0,C 180,E1 -10985.999,E2 -10985.999} C_VEL
LIN {X 0,Y 407.285,Z 445.573,A -85,B 0,C 180,E1 -10986.565,E2 -10986.565} C_VEL
LIN {X 0,Y 406.776,Z 455.855,A -85,B 0,C 180,E1 -10987.321,E2 -10987.321} C_VEL
LIN {X 0,Y 406.215,Z 464.109,A -85,B 0,C 180,E1 -10988.076,E2 -10988.076} C_VEL
LIN {X 0,Y 405.621,Z 472.116,A -85,B 0,C 180,E1 -10988.972,E2 -10988.972} C_VEL
LIN {X 0,Y 405.102,Z 479.571,A -85,B 0,C 180,E1 -10989.991,E2 -10989.991} C_VEL
LIN {X 0,Y 404.55,Z 487.166,A -85,B 0,C 180,E1 -10991.271,E2 -10991.271} C_VEL
LIN {X 0,Y 404.076,Z 492.965,A -85,B 0,C 180,E1 -10992.518,E2 -10992.518} C_VEL
LIN {X 0,Y 403.751,Z 497.025,A -85,B 0,C 180,E1 -10993.592,E2 -10993.592} C_VEL
LIN {X 0,Y 403.507,Z 500.19,A -85,B 0,C 180,E1 -10994.629,E2 -10994.629} C_VEL
LIN {X 0,Y 403.225,Z 503.676,A -85,B 0,C 180,E1 -10996.193,E2 -10996.193} C_VEL
LIN {X 0,Y 403.058,Z 505.318,A -85,B 0,C 180,E1 -10997.244,E2 -10997.244} C_VEL
LIN {X 0,Y 402.928,Z 506.313,A -85,B 0,C 180,E1 -10998.299,E2 -10998.299} C_VEL
LIN {X 0,Y 402.892,Z 506.779,A -85,B 0,C 180,E1 -10999.625,E2 -10999.625} C_VEL
LIN {X 0,Y 402.886,Z 505.841,A -85,B 0,C 180,E1 -11001.49,E2 -11001.49} C_VEL
LIN {X 0,Y 402.976,Z 504.54,A -85,B 0,C 180,E1 -11002.563,E2 -11002.563} C_VEL
LIN {X 0,Y 403.124,Z 502.606,A -85,B 0,C 180,E1 -11003.64,E2 -11003.64} C_VEL
LIN {X 0,Y 403.288,Z 499.075,A -85,B 0,C 180,E1 -11005.023,E2 -11005.023} C_VEL
LIN {X 0,Y 403.482,Z 494.467,A -85,B 0,C 180,E1 -11006.371,E2 -11006.371} C_VEL
LIN {X 0,Y 403.796,Z 488.953,A -85,B 0,C 180,E1 -11007.634,E2 -11007.634} C_VEL
LIN {X 0,Y 404.15,Z 482.33,A -85,B 0,C 180,E1 -11008.853,E2 -11008.853} C_VEL
LIN {X 0,Y 404.64,Z 474.094,A -85,B 0,C 180,E1 -11010.076,E2 -11010.076} C_VEL
LIN {X 0,Y 405.128,Z 464.164,A -85,B 0,C 180,E1 -11011.216,E2 -11011.216} C_VEL
LIN {X 0,Y 405.557,Z 456.331,A -85,B 0,C 180,E1 -11011.943,E2 -11011.943} C_VEL
LIN {X 0,Y 405.905,Z 447.503,A -85,B 0,C 180,E1 -11012.61,E2 -11012.61} C_VEL
LIN {X 0,Y 406.292,Z 438.127,A -85,B 0,C 180,E1 -11013.165,E2 -11013.165} C_VEL
LIN {X 0,Y 406.567,Z 427.755,A -85,B 0,C 180,E1 -11013.623,E2 -11013.623} C_VEL
LIN {X 0,Y 406.873,Z 413.272,A -85,B 0,C 180,E1 -11014.015,E2 -11014.015} C_VEL
LIN {X 0,Y 407.665,Z 357.99,A -85,B 0,C 180,E1 -11015.18,E2 -11015.18} C_VEL
LIN {X 0,Y 404.885,Z 339.291,A -85,B 0,C 180,E1 -11015.7,E2 -11015.7} C_VEL
LIN {X 0,Y 405.695,Z 323.637,A -85,B 0,C 180,E1 -11018.97,E2 -11018.97} C_VEL
LIN {X 0,Y 406.548,Z 307.607,A -85,B 0,C 180,E1 -11022.392,E2 -11022.392} C_VEL
LIN {X 0,Y 406.608,Z 302.743,A -85,B 0,C 180,E1 -11023.455,E2 -11023.455} C_VEL
LIN {X 0,Y 404.152,Z 290.141,A -85,B 0,C 180,E1 -11026.436,E2 -11026.436} C_VEL
LIN {X 0,Y 404.127,Z 290.144,A -85,B 0,C 180,E1 -11029.953,E2 -11029.953} C_VEL
LIN {X 0,Y 404.128,Z 290.142,A -85,B 0,C 180,E1 -11033.128,E2 -11033.128} C_VEL
LIN {X 0,Y 404.136,Z 290.142,A -85,B 0,C 180,E1 -11036.188,E2 -11036.188} C_VEL
LIN {X 0,Y 404.142,Z 290.143,A -85,B 0,C 180,E1 -11039.716,E2 -11039.716} C_VEL
LIN {X 0,Y 404.104,Z 290.143,A -85,B 0,C 180,E1 -11043.117,E2 -11043.117} C_VEL
LIN {X 0,Y 404.149,Z 290.145,A -85,B 0,C 180,E1 -11046.425,E2 -11046.425} C_VEL
LIN {X 0,Y 404.159,Z 290.137,A -85,B 0,C 180,E1 -11049.889,E2 -11049.889} C_VEL
LIN {X 0,Y 404.221,Z 290.133,A -85,B 0,C 180,E1 -11052.993,E2 -11052.993} C_VEL
LIN {X 0,Y 404.289,Z 290.128,A -85,B 0,C 180,E1 -11056.938,E2 -11056.938} C_VEL
LIN {X 0,Y 404.253,Z 290.125,A -85,B 0,C 180,E1 -11059.987,E2 -11059.987} C_VEL
LIN {X 0,Y 404.345,Z 290.117,A -85,B 0,C 180,E1 -11063.01,E2 -11063.01} C_VEL
LIN {X 0,Y 404.36,Z 290.112,A -85,B 0,C 180,E1 -11063.872,E2 -11063.872} C_VEL
LIN {X 0,Y 403.763,Z 290.189,A -85,B 0,C 180,E1 -11064.702,E2 -11064.702} C_VEL
LIN {X 0,Y 401.003,Z 290.536,A -85,B 0,C 180,E1 -11066.053,E2 -11066.053} C_VEL
LIN {X 0,Y 398.598,Z 290.835,A -85,B 0,C 180,E1 -11067.143,E2 -11067.143} C_VEL
LIN {X 0,Y 397.51,Z 290.968,A -85,B 0,C 180,E1 -11067.985,E2 -11067.985} C_VEL
LIN {X 0,Y 397.394,Z 290.98,A -85,B 0,C 180,E1 -11068.271,E2 -11068.271} C_VEL
LIN {X 0,Y 397.441,Z 290.979,A -85,B 0,C 180,E1 -11072.025,E2 -11072.025} C_VEL
LIN {X 0,Y 397.321,Z 290.996,A -85,B 0,C 180,E1 -11076.09,E2 -11076.09} C_VEL
LIN {X 0,Y 397.229,Z 290.999,A -85,B 0,C 180,E1 -11079.159,E2 -11079.159} C_VEL
LIN {X 0,Y 397.217,Z 291.007,A -85,B 0,C 180,E1 -11082.255,E2 -11082.255} C_VEL
LIN {X 0,Y 397.175,Z 291.007,A -85,B 0,C 180,E1 -11085.388,E2 -11085.388} C_VEL
LIN {X 0,Y 397.153,Z 291.014,A -85,B 0,C 180,E1 -11088.57,E2 -11088.57} C_VEL
LIN {X 0,Y 397.088,Z 291.017,A -85,B 0,C 180,E1 -11091.814,E2 -11091.814} C_VEL
LIN {X 0,Y 397.091,Z 291.024,A -85,B 0,C 180,E1 -11095.131,E2 -11095.131} C_VEL
LIN {X 0,Y 397.06,Z 291.021,A -85,B 0,C 180,E1 -11098.543,E2 -11098.543} C_VEL
LIN {X 0,Y 397.066,Z 291.024,A -85,B 0,C 180,E1 -11101.832,E2 -11101.832} C_VEL
LIN {X 0,Y 397.107,Z 291.015,A -85,B 0,C 180,E1 -11104.489,E2 -11104.489} C_VEL
LIN {X 0,Y 397.076,Z 291.022,A -85,B 0,C 180,E1 -11108.271,E2 -11108.271} C_VEL
LIN {X 0,Y 397.039,Z 291.023,A -85,B 0,C 180,E1 -11110.907,E2 -11110.907} C_VEL
LIN {X 0,Y 397.073,Z 291.02,A -85,B 0,C 180,E1 -11113.644,E2 -11113.644} C_VEL
LIN {X 0,Y 397.072,Z 291.025,A -85,B 0,C 180,E1 -11116.516,E2 -11116.516} C_VEL
LIN {X 0,Y 397.081,Z 291.023,A -85,B 0,C 180,E1 -11120.418,E2 -11120.418} C_VEL
LIN {X 0,Y 397.062,Z 291.025,A -85,B 0,C 180,E1 -11123,E2 -11123} C_VEL
LIN {X 0,Y 397.073,Z 291.023,A -85,B 0,C 180,E1 -11126.722,E2 -11126.722} C_VEL
LIN {X 0,Y 397.09,Z 291.017,A -85,B 0,C 180,E1 -11130.292,E2 -11130.292} C_VEL
LIN {X 0,Y 397.152,Z 291.01,A -85,B 0,C 180,E1 -11132.606,E2 -11132.606} C_VEL
LIN {X 0,Y 397.083,Z 291.02,A -85,B 0,C 180,E1 -11135.978,E2 -11135.978} C_VEL
LIN {X 0,Y 397.07,Z 291.027,A -85,B 0,C 180,E1 -11139.71,E2 -11139.71} C_VEL
LIN {X 0,Y 397.133,Z 291.011,A -85,B 0,C 180,E1 -11142.843,E2 -11142.843} C_VEL
LIN {X 0,Y 397.179,Z 291.007,A -85,B 0,C 180,E1 -11146.7,E2 -11146.7} C_VEL
LIN {X 0,Y 397.174,Z 291.008,A -85,B 0,C 180,E1 -11149.807,E2 -11149.807} C_VEL
LIN {X 0,Y 397.302,Z 290.993,A -85,B 0,C 180,E1 -11152.887,E2 -11152.887} C_VEL
LIN {X 0,Y 397.204,Z 291.006,A -85,B 0,C 180,E1 -11154.924,E2 -11154.924} C_VEL
LIN {X 0,Y 397.397,Z 290.979,A -85,B 0,C 180,E1 -11157.972,E2 -11157.972} C_VEL
LIN {X 0,Y 397.524,Z 290.963,A -85,B 0,C 180,E1 -11159.999,E2 -11159.999} C_VEL
LIN {X 0,Y 397.332,Z 290.995,A -85,B 0,C 180,E1 -11163.041,E2 -11163.041} C_VEL
LIN {X 0,Y 397.301,Z 290.996,A -85,B 0,C 180,E1 -11167.112,E2 -11167.112} C_VEL
LIN {X 0,Y 397.166,Z 291.008,A -85,B 0,C 180,E1 -11170.192,E2 -11170.192} C_VEL
LIN {X 0,Y 397.175,Z 291.01,A -85,B 0,C 180,E1 -11173.322,E2 -11173.322} C_VEL
LIN {X 0,Y 397.131,Z 291.012,A -85,B 0,C 180,E1 -11177.156,E2 -11177.156} C_VEL
LIN {X 0,Y 397.054,Z 291.022,A -85,B 0,C 180,E1 -11180.732,E2 -11180.732} C_VEL
LIN {X 0,Y 397.085,Z 291.022,A -85,B 0,C 180,E1 -11184.021,E2 -11184.021} C_VEL
LIN {X 0,Y 397.147,Z 291.01,A -85,B 0,C 180,E1 -11187.393,E2 -11187.393} C_VEL
LIN {X 0,Y 397.033,Z 291.029,A -85,B 0,C 180,E1 -11190.886,E2 -11190.886} C_VEL
LIN {X 0,Y 397.083,Z 291.021,A -85,B 0,C 180,E1 -11194.497,E2 -11194.497} C_VEL
LIN {X 0,Y 397.06,Z 291.021,A -85,B 0,C 180,E1 -11198.279,E2 -11198.279} C_VEL
LIN {X 0,Y 397.05,Z 291.026,A -85,B 0,C 180,E1 -11200.913,E2 -11200.913} C_VEL
LIN {X 0,Y 397.065,Z 291.024,A -85,B 0,C 180,E1 -11203.653,E2 -11203.653} C_VEL
LIN {X 0,Y 397.069,Z 291.019,A -85,B 0,C 180,E1 -11206.525,E2 -11206.525} C_VEL
LIN {X 0,Y 397.072,Z 291.025,A -85,B 0,C 180,E1 -11209.559,E2 -11209.559} C_VEL
LIN {X 0,Y 397.067,Z 291.02,A -85,B 0,C 180,E1 -11213.008,E2 -11213.008} C_VEL
LIN {X 0,Y 397.088,Z 291.018,A -85,B 0,C 180,E1 -11216.731,E2 -11216.731} C_VEL
LIN {X 0,Y 397.095,Z 291.021,A -85,B 0,C 180,E1 -11220.299,E2 -11220.299} C_VEL
LIN {X 0,Y 397.117,Z 291.046,A -85,B 0,C 180,E1 -11221.173,E2 -11221.173} C_VEL
LIN {X 0,Y 400.919,Z 308.369,A -85,B 0,C 180,E1 -11224.571,E2 -11224.571} C_VEL
LIN {X 0,Y 401.555,Z 311.504,A -85,B 0,C 180,E1 -11225.167,E2 -11225.167} C_VEL
LIN {X 0,Y 400.99,Z 320.699,A -85,B 0,C 180,E1 -11226.779,E2 -11226.779} C_VEL
LIN {X 0,Y 399.436,Z 340.585,A -85,B 0,C 180,E1 -11230.207,E2 -11230.207} C_VEL
LIN {X 0,Y 399.17,Z 344.807,A -85,B 0,C 180,E1 -11230.905,E2 -11230.905} C_VEL
LIN {X 0,Y 401.846,Z 368.437,A -85,B 0,C 180,E1 -11231.489,E2 -11231.489} C_VEL
LIN {X 0,Y 400.586,Z 450.084,A -85,B 0,C 180,E1 -11233.111,E2 -11233.111} C_VEL
LIN {X 0,Y 400.244,Z 459.105,A -85,B 0,C 180,E1 -11233.392,E2 -11233.392} C_VEL
LIN {X 0,Y 399.844,Z 468.641,A -85,B 0,C 180,E1 -11233.801,E2 -11233.801} C_VEL
LIN {X 0,Y 399.438,Z 477.76,A -85,B 0,C 180,E1 -11234.309,E2 -11234.309} C_VEL
LIN {X 0,Y 398.822,Z 488.405,A -85,B 0,C 180,E1 -11235.069,E2 -11235.069} C_VEL
LIN {X 0,Y 398.318,Z 497.9,A -85,B 0,C 180,E1 -11235.914,E2 -11235.914} C_VEL
LIN {X 0,Y 397.75,Z 506.633,A -85,B 0,C 180,E1 -11236.854,E2 -11236.854} C_VEL
LIN {X 0,Y 397.212,Z 515.439,A -85,B 0,C 180,E1 -11238.004,E2 -11238.004} C_VEL
LIN {X 0,Y 396.764,Z 522.052,A -85,B 0,C 180,E1 -11239.026,E2 -11239.026} C_VEL
LIN {X 0,Y 396.395,Z 528.968,A -85,B 0,C 180,E1 -11240.306,E2 -11240.306} C_VEL
LIN {X 0,Y 396.185,Z 533.711,A -85,B 0,C 180,E1 -11241.331,E2 -11241.331} C_VEL
LIN {X 0,Y 395.993,Z 539.457,A -85,B 0,C 180,E1 -11242.866,E2 -11242.866} C_VEL
LIN {X 0,Y 395.843,Z 543.364,A -85,B 0,C 180,E1 -11244.169,E2 -11244.169} C_VEL
LIN {X 0,Y 395.817,Z 547.249,A -85,B 0,C 180,E1 -11245.93,E2 -11245.93} C_VEL
LIN {X 0,Y 395.868,Z 548.886,A -85,B 0,C 180,E1 -11246.949,E2 -11246.949} C_VEL
LIN {X 0,Y 395.871,Z 550.825,A -85,B 0,C 180,E1 -11248.985,E2 -11248.985} C_VEL
LIN {X 0,Y 395.874,Z 551.112,A -85,B 0,C 180,E1 -11250.002,E2 -11250.002} C_VEL
LIN {X 0,Y 395.901,Z 550.496,A -85,B 0,C 180,E1 -11252.037,E2 -11252.037} C_VEL
LIN {X 0,Y 395.807,Z 548.021,A -85,B 0,C 180,E1 -11254.074,E2 -11254.074} C_VEL
LIN {X 0,Y 395.868,Z 546.252,A -85,B 0,C 180,E1 -11255.094,E2 -11255.094} C_VEL
LIN {X 0,Y 395.926,Z 542.715,A -85,B 0,C 180,E1 -11256.576,E2 -11256.576} C_VEL
LIN {X 0,Y 396.098,Z 537.723,A -85,B 0,C 180,E1 -11258.162,E2 -11258.162} C_VEL
LIN {X 0,Y 396.429,Z 531.555,A -85,B 0,C 180,E1 -11259.697,E2 -11259.697} C_VEL
LIN {X 0,Y 396.845,Z 525.294,A -85,B 0,C 180,E1 -11260.976,E2 -11260.976} C_VEL
LIN {X 0,Y 397.473,Z 517.729,A -85,B 0,C 180,E1 -11262.251,E2 -11262.251} C_VEL
LIN {X 0,Y 398.056,Z 509.334,A -85,B 0,C 180,E1 -11263.426,E2 -11263.426} C_VEL
LIN {X 0,Y 398.749,Z 500.821,A -85,B 0,C 180,E1 -11264.416,E2 -11264.416} C_VEL
LIN {X 0,Y 399.459,Z 491.658,A -85,B 0,C 180,E1 -11265.303,E2 -11265.303} C_VEL
LIN {X 0,Y 400.175,Z 482.131,A -85,B 0,C 180,E1 -11266.058,E2 -11266.058} C_VEL
LIN {X 0,Y 400.848,Z 472.264,A -85,B 0,C 180,E1 -11266.685,E2 -11266.685} C_VEL
LIN {X 0,Y 401.45,Z 461.302,A -85,B 0,C 180,E1 -11267.216,E2 -11267.216} C_VEL
LIN {X 0,Y 401.864,Z 451.677,A -85,B 0,C 180,E1 -11267.559,E2 -11267.559} C_VEL
LIN {X 0,Y 402.33,Z 433.298,A -85,B 0,C 180,E1 -11267.965,E2 -11267.965} C_VEL
LIN {X 0,Y 403.462,Z 366.098,A -85,B 0,C 180,E1 -11269.342,E2 -11269.342} C_VEL
LIN {X 0,Y 400.473,Z 345.356,A -85,B 0,C 180,E1 -11269.989,E2 -11269.989} C_VEL
LIN {X 0,Y 400.216,Z 343.729,A -85,B 0,C 180,E1 -11270.048,E2 -11270.048} C_VEL
LIN {X 0,Y 401.68,Z 322.635,A -85,B 0,C 180,E1 -11273.456,E2 -11273.456} C_VEL
LIN {X 0,Y 402.308,Z 312.795,A -85,B 0,C 180,E1 -11275.063,E2 -11275.063} C_VEL
LIN {X 0,Y 399.887,Z 301.534,A -85,B 0,C 180,E1 -11277.19,E2 -11277.19} C_VEL
LIN {X 0,Y 397.116,Z 291.028,A -85,B 0,C 180,E1 -11279.303,E2 -11279.303} C_VEL
LIN {X 0,Y 397.107,Z 291.022,A -85,B 0,C 180,E1 -11283.272,E2 -11283.272} C_VEL
LIN {X 0,Y 397.099,Z 291.025,A -85,B 0,C 180,E1 -11285.734,E2 -11285.734} C_VEL
LIN {X 0,Y 397.104,Z 291.024,A -85,B 0,C 180,E1 -11289.576,E2 -11289.576} C_VEL
LIN {X 0,Y 397.092,Z 291.023,A -85,B 0,C 180,E1 -11293.478,E2 -11293.478} C_VEL
LIN {X 0,Y 397.09,Z 291.022,A -85,B 0,C 180,E1 -11296.52,E2 -11296.52} C_VEL
LIN {X 0,Y 397.104,Z 291.021,A -85,B 0,C 180,E1 -11299.551,E2 -11299.551} C_VEL
LIN {X 0,Y 397.081,Z 291.019,A -85,B 0,C 180,E1 -11302.789,E2 -11302.789} C_VEL
LIN {X 0,Y 397.1,Z 291.016,A -85,B 0,C 180,E1 -11306.281,E2 -11306.281} C_VEL
LIN {X 0,Y 397.092,Z 291.015,A -85,B 0,C 180,E1 -11310.133,E2 -11310.133} C_VEL
LIN {X 0,Y 397.174,Z 291.01,A -85,B 0,C 180,E1 -11312.609,E2 -11312.609} C_VEL
LIN {X 0,Y 397.114,Z 291.018,A -85,B 0,C 180,E1 -11315.981,E2 -11315.981} C_VEL
LIN {X 0,Y 397.132,Z 291.016,A -85,B 0,C 180,E1 -11319.272,E2 -11319.272} C_VEL
LIN {X 0,Y 397.158,Z 291.014,A -85,B 0,C 180,E1 -11322.845,E2 -11322.845} C_VEL
LIN {X 0,Y 397.205,Z 291.009,A -85,B 0,C 180,E1 -11326.702,E2 -11326.702} C_VEL
LIN {X 0,Y 397.197,Z 291.011,A -85,B 0,C 180,E1 -11329.809,E2 -11329.809} C_VEL
LIN {X 0,Y 397.321,Z 291,A -85,B 0,C 180,E1 -11332.888,E2 -11332.888} C_VEL
LIN {X 0,Y 397.248,Z 291.192,A -85,B 0,C 180,E1 -11334.989,E2 -11334.989} C_VEL
LIN {X 0,Y 400.189,Z 301.632,A -85,B 0,C 180,E1 -11336.981,E2 -11336.981} C_VEL
LIN {X 0,Y 400.334,Z 306.163,A -85,B 0,C 180,E1 -11337.737,E2 -11337.737} C_VEL
LIN {X 0,Y 399.452,Z 327.984,A -85,B 0,C 180,E1 -11341.261,E2 -11341.261} C_VEL
LIN {X 0,Y 399.193,Z 338.222,A -85,B 0,C 180,E1 -11342.902,E2 -11342.902} C_VEL
LIN {X 0,Y 402.953,Z 359.225,A -85,B 0,C 180,E1 -11343.674,E2 -11343.674} C_VEL
LIN {X 0,Y 402.597,Z 378.734,A -85,B 0,C 180,E1 -11344.143,E2 -11344.143} C_VEL
LIN {X 0,Y 401.473,Z 423.333,A -85,B 0,C 180,E1 -11345.211,E2 -11345.211} C_VEL
LIN {X 0,Y 401.04,Z 434.484,A -85,B 0,C 180,E1 -11345.626,E2 -11345.626} C_VEL
LIN {X 0,Y 400.498,Z 446.52,A -85,B 0,C 180,E1 -11346.297,E2 -11346.297} C_VEL
LIN {X 0,Y 399.959,Z 456.645,A -85,B 0,C 180,E1 -11347.066,E2 -11347.066} C_VEL
LIN {X 0,Y 399.371,Z 464.847,A -85,B 0,C 180,E1 -11347.839,E2 -11347.839} C_VEL
LIN {X 0,Y 398.656,Z 473.795,A -85,B 0,C 180,E1 -11348.877,E2 -11348.877} C_VEL
LIN {X 0,Y 397.989,Z 482.614,A -85,B 0,C 180,E1 -11350.172,E2 -11350.172} C_VEL
LIN {X 0,Y 397.412,Z 489.555,A -85,B 0,C 180,E1 -11351.476,E2 -11351.476} C_VEL
LIN {X 0,Y 396.956,Z 494.719,A -85,B 0,C 180,E1 -11352.68,E2 -11352.68} C_VEL
LIN {X 0,Y 396.636,Z 498.709,A -85,B 0,C 180,E1 -11353.84,E2 -11353.84} C_VEL
LIN {X 0,Y 396.403,Z 501.623,A -85,B 0,C 180,E1 -11354.897,E2 -11354.897} C_VEL
LIN {X 0,Y 396.09,Z 505.012,A -85,B 0,C 180,E1 -11356.647,E2 -11356.647} C_VEL
LIN {X 0,Y 395.947,Z 506.141,A -85,B 0,C 180,E1 -11357.563,E2 -11357.563} C_VEL
LIN {X 0,Y 395.828,Z 506.961,A -85,B 0,C 180,E1 -11358.639,E2 -11358.639} C_VEL
LIN {X 0,Y 395.795,Z 507.196,A -85,B 0,C 180,E1 -11359.772,E2 -11359.772} C_VEL
LIN {X 0,Y 395.774,Z 506.791,A -85,B 0,C 180,E1 -11360.803,E2 -11360.803} C_VEL
LIN {X 0,Y 395.904,Z 504.811,A -85,B 0,C 180,E1 -11362.626,E2 -11362.626} C_VEL
LIN {X 0,Y 396.075,Z 501.959,A -85,B 0,C 180,E1 -11364.087,E2 -11364.087} C_VEL
LIN {X 0,Y 396.227,Z 498.895,A -85,B 0,C 180,E1 -11365.238,E2 -11365.238} C_VEL
LIN {X 0,Y 396.526,Z 493.103,A -85,B 0,C 180,E1 -11366.87,E2 -11366.87} C_VEL
LIN {X 0,Y 396.899,Z 486.43,A -85,B 0,C 180,E1 -11368.309,E2 -11368.309} C_VEL
LIN {X 0,Y 397.356,Z 478.05,A -85,B 0,C 180,E1 -11369.686,E2 -11369.686} C_VEL
LIN {X 0,Y 397.729,Z 471.397,A -85,B 0,C 180,E1 -11370.582,E2 -11370.582} C_VEL
LIN {X 0,Y 398.142,Z 464.316,A -85,B 0,C 180,E1 -11371.382,E2 -11371.382} C_VEL
LIN {X 0,Y 398.613,Z 455.575,A -85,B 0,C 180,E1 -11372.195,E2 -11372.195} C_VEL
LIN {X 0,Y 398.969,Z 447.406,A -85,B 0,C 180,E1 -11372.811,E2 -11372.811} C_VEL
LIN {X 0,Y 399.335,Z 438.136,A -85,B 0,C 180,E1 -11373.366,E2 -11373.366} C_VEL
LIN {X 0,Y 399.645,Z 426.85,A -85,B 0,C 180,E1 -11373.866,E2 -11373.866} C_VEL
LIN {X 0,Y 399.979,Z 412.17,A -85,B 0,C 180,E1 -11374.248,E2 -11374.248} C_VEL
LIN {X 0,Y 400.713,Z 358.593,A -85,B 0,C 180,E1 -11375.405,E2 -11375.405} C_VEL
LIN {X 0,Y 397.925,Z 339.337,A -85,B 0,C 180,E1 -11375.947,E2 -11375.947} C_VEL
LIN {X 0,Y 398.729,Z 324.238,A -85,B 0,C 180,E1 -11379.149,E2 -11379.149} C_VEL
LIN {X 0,Y 399.54,Z 309.314,A -85,B 0,C 180,E1 -11382.375,E2 -11382.375} C_VEL
LIN {X 0,Y 399.638,Z 303.917,A -85,B 0,C 180,E1 -11383.574,E2 -11383.574} C_VEL
LIN {X 0,Y 397.104,Z 291.021,A -85,B 0,C 180,E1 -11386.657,E2 -11386.657} C_VEL
LIN {X 0,Y 397.081,Z 291.019,A -85,B 0,C 180,E1 -11390.421,E2 -11390.421} C_VEL
LIN {X 0,Y 397.09,Z 291.018,A -85,B 0,C 180,E1 -11393.006,E2 -11393.006} C_VEL
LIN {X 0,Y 397.11,Z 291.014,A -85,B 0,C 180,E1 -11396.728,E2 -11396.728} C_VEL
LIN {X 0,Y 397.115,Z 291.018,A -85,B 0,C 180,E1 -11400.296,E2 -11400.296} C_VEL
LIN {X 0,Y 397.076,Z 291.021,A -85,B 0,C 180,E1 -11403.738,E2 -11403.738} C_VEL
LIN {X 0,Y 397.102,Z 291.016,A -85,B 0,C 180,E1 -11407.085,E2 -11407.085} C_VEL
LIN {X 0,Y 397.135,Z 291.016,A -85,B 0,C 180,E1 -11410.352,E2 -11410.352} C_VEL
LIN {X 0,Y 397.168,Z 291.007,A -85,B 0,C 180,E1 -11413.553,E2 -11413.553} C_VEL
LIN {X 0,Y 397.235,Z 291.003,A -85,B 0,C 180,E1 -11416.702,E2 -11416.702} C_VEL
LIN {X 0,Y 397.214,Z 291.002,A -85,B 0,C 180,E1 -11419.808,E2 -11419.808} C_VEL
LIN {X 0,Y 397.298,Z 290.993,A -85,B 0,C 180,E1 -11422.886,E2 -11422.886} C_VEL
LIN {X 0,Y 397.23,Z 291.001,A -85,B 0,C 180,E1 -11424.923,E2 -11424.923} C_VEL
LIN {X 0,Y 397.394,Z 290.98,A -85,B 0,C 180,E1 -11428.271,E2 -11428.271} C_VEL
LIN {X 0,Y 396.669,Z 291.072,A -85,B 0,C 180,E1 -11429.116,E2 -11429.116} C_VEL
LIN {X 0,Y 393.848,Z 291.421,A -85,B 0,C 180,E1 -11430.492,E2 -11430.492} C_VEL
LIN {X 0,Y 391.467,Z 291.722,A -85,B 0,C 180,E1 -11431.603,E2 -11431.603} C_VEL
LIN {X 0,Y 390.395,Z 291.852,A -85,B 0,C 180,E1 -11432.46,E2 -11432.46} C_VEL
LIN {X 0,Y 390.279,Z 291.865,A -85,B 0,C 180,E1 -11432.751,E2 -11432.751} C_VEL
LIN {X 0,Y 390.277,Z 291.872,A -85,B 0,C 180,E1 -11436.2,E2 -11436.2} C_VEL
LIN {X 0,Y 390.188,Z 291.876,A -85,B 0,C 180,E1 -11439.326,E2 -11439.326} C_VEL
LIN {X 0,Y 390.169,Z 291.887,A -85,B 0,C 180,E1 -11442.48,E2 -11442.48} C_VEL
LIN {X 0,Y 390.135,Z 291.883,A -85,B 0,C 180,E1 -11445.673,E2 -11445.673} C_VEL
LIN {X 0,Y 390.097,Z 291.894,A -85,B 0,C 180,E1 -11448.918,E2 -11448.918} C_VEL
LIN {X 0,Y 390.029,Z 291.897,A -85,B 0,C 180,E1 -11452.23,E2 -11452.23} C_VEL
LIN {X 0,Y 390.04,Z 291.897,A -85,B 0,C 180,E1 -11455.718,E2 -11455.718} C_VEL
LIN {X 0,Y 390.017,Z 291.902,A -85,B 0,C 180,E1 -11459.107,E2 -11459.107} C_VEL
LIN {X 0,Y 390.026,Z 291.897,A -85,B 0,C 180,E1 -11462.717,E2 -11462.717} C_VEL
LIN {X 0,Y 390.036,Z 291.903,A -85,B 0,C 180,E1 -11465.82,E2 -11465.82} C_VEL
LIN {X 0,Y 390.043,Z 291.895,A -85,B 0,C 180,E1 -11469.213,E2 -11469.213} C_VEL
LIN {X 0,Y 390.03,Z 291.896,A -85,B 0,C 180,E1 -11473.206,E2 -11473.206} C_VEL
LIN {X 0,Y 390.027,Z 291.9,A -85,B 0,C 180,E1 -11476.785,E2 -11476.785} C_VEL
LIN {X 0,Y 390.025,Z 291.897,A -85,B 0,C 180,E1 -11479.556,E2 -11479.556} C_VEL
LIN {X 0,Y 390.008,Z 291.903,A -85,B 0,C 180,E1 -11482.445,E2 -11482.445} C_VEL
LIN {X 0,Y 390.024,Z 291.897,A -85,B 0,C 180,E1 -11486.04,E2 -11486.04} C_VEL
LIN {X 0,Y 390.01,Z 291.899,A -85,B 0,C 180,E1 -11489.864,E2 -11489.864} C_VEL
LIN {X 0,Y 390.07,Z 291.897,A -85,B 0,C 180,E1 -11493.228,E2 -11493.228} C_VEL
LIN {X 0,Y 390.022,Z 291.897,A -85,B 0,C 180,E1 -11496.761,E2 -11496.761} C_VEL
LIN {X 0,Y 390.038,Z 291.9,A -85,B 0,C 180,E1 -11499.979,E2 -11499.979} C_VEL
LIN {X 0,Y 390.088,Z 291.89,A -85,B 0,C 180,E1 -11503.245,E2 -11503.245} C_VEL
LIN {X 0,Y 390.145,Z 291.884,A -85,B 0,C 180,E1 -11506.559,E2 -11506.559} C_VEL
LIN {X 0,Y 390.124,Z 291.885,A -85,B 0,C 180,E1 -11509.621,E2 -11509.621} C_VEL
LIN {X 0,Y 390.254,Z 291.873,A -85,B 0,C 180,E1 -11512.757,E2 -11512.757} C_VEL
LIN {X 0,Y 390.176,Z 291.883,A -85,B 0,C 180,E1 -11514.832,E2 -11514.832} C_VEL
LIN {X 0,Y 390.367,Z 291.854,A -85,B 0,C 180,E1 -11517.936,E2 -11517.936} C_VEL
LIN {X 0,Y 390.494,Z 291.838,A -85,B 0,C 180,E1 -11519.999,E2 -11519.999} C_VEL
LIN {X 0,Y 390.266,Z 291.875,A -85,B 0,C 180,E1 -11523.096,E2 -11523.096} C_VEL
LIN {X 0,Y 390.274,Z 291.866,A -85,B 0,C 180,E1 -11526.202,E2 -11526.202} C_VEL
LIN {X 0,Y 390.152,Z 291.888,A -85,B 0,C 180,E1 -11529.33,E2 -11529.33} C_VEL
LIN {X 0,Y 390.124,Z 291.884,A -85,B 0,C 180,E1 -11532.484,E2 -11532.484} C_VEL
LIN {X 0,Y 390.086,Z 291.896,A -85,B 0,C 180,E1 -11535.678,E2 -11535.678} C_VEL
LIN {X 0,Y 390.053,Z 291.893,A -85,B 0,C 180,E1 -11538.924,E2 -11538.924} C_VEL
LIN {X 0,Y 389.993,Z 291.908,A -85,B 0,C 180,E1 -11542.236,E2 -11542.236} C_VEL
LIN {X 0,Y 390.071,Z 291.892,A -85,B 0,C 180,E1 -11545.745,E2 -11545.745} C_VEL
LIN {X 0,Y 390.007,Z 291.901,A -85,B 0,C 180,E1 -11549.113,E2 -11549.113} C_VEL
LIN {X 0,Y 389.999,Z 291.908,A -85,B 0,C 180,E1 -11552.725,E2 -11552.725} C_VEL
LIN {X 0,Y 390.014,Z 291.898,A -85,B 0,C 180,E1 -11555.828,E2 -11555.828} C_VEL
LIN {X 0,Y 390.024,Z 291.904,A -85,B 0,C 180,E1 -11559.22,E2 -11559.22} C_VEL
LIN {X 0,Y 390.002,Z 291.9,A -85,B 0,C 180,E1 -11562.377,E2 -11562.377} C_VEL
LIN {X 0,Y 390.009,Z 291.905,A -85,B 0,C 180,E1 -11565.358,E2 -11565.358} C_VEL
LIN {X 0,Y 389.998,Z 291.902,A -85,B 0,C 180,E1 -11568.19,E2 -11568.19} C_VEL
LIN {X 0,Y 390.034,Z 291.896,A -85,B 0,C 180,E1 -11570.908,E2 -11570.908} C_VEL
LIN {X 0,Y 390.043,Z 291.895,A -85,B 0,C 180,E1 -11574.795,E2 -11574.795} C_VEL
LIN {X 0,Y 389.999,Z 291.905,A -85,B 0,C 180,E1 -11578.499,E2 -11578.499} C_VEL
LIN {X 0,Y 390.079,Z 292.009,A -85,B 0,C 180,E1 -11580.898,E2 -11580.898} C_VEL
LIN {X 0,Y 393.519,Z 307.791,A -85,B 0,C 180,E1 -11584.057,E2 -11584.057} C_VEL
LIN {X 0,Y 394.674,Z 313.964,A -85,B 0,C 180,E1 -11585.251,E2 -11585.251} C_VEL
LIN {X 0,Y 393.088,Z 333.413,A -85,B 0,C 180,E1 -11588.687,E2 -11588.687} C_VEL
LIN {X 0,Y 392.219,Z 344.557,A -85,B 0,C 180,E1 -11590.637,E2 -11590.637} C_VEL
LIN {X 0,Y 394.946,Z 369.069,A -85,B 0,C 180,E1 -11591.255,E2 -11591.255} C_VEL
LIN {X 0,Y 393.649,Z 449.934,A -85,B 0,C 180,E1 -11592.905,E2 -11592.905} C_VEL
LIN {X 0,Y 393.282,Z 459.717,A -85,B 0,C 180,E1 -11593.223,E2 -11593.223} C_VEL
LIN {X 0,Y 392.861,Z 469.003,A -85,B 0,C 180,E1 -11593.639,E2 -11593.639} C_VEL
LIN {X 0,Y 392.437,Z 477.975,A -85,B 0,C 180,E1 -11594.155,E2 -11594.155} C_VEL
LIN {X 0,Y 391.808,Z 488.52,A -85,B 0,C 180,E1 -11594.928,E2 -11594.928} C_VEL
LIN {X 0,Y 391.358,Z 496.486,A -85,B 0,C 180,E1 -11595.636,E2 -11595.636} C_VEL
LIN {X 0,Y 390.704,Z 506.622,A -85,B 0,C 180,E1 -11596.745,E2 -11596.745} C_VEL
LIN {X 0,Y 390.171,Z 514.511,A -85,B 0,C 180,E1 -11597.784,E2 -11597.784} C_VEL
LIN {X 0,Y 389.759,Z 521.232,A -85,B 0,C 180,E1 -11598.826,E2 -11598.826} C_VEL
LIN {X 0,Y 389.355,Z 528.232,A -85,B 0,C 180,E1 -11600.129,E2 -11600.129} C_VEL
LIN {X 0,Y 389.092,Z 534.045,A -85,B 0,C 180,E1 -11601.433,E2 -11601.433} C_VEL
LIN {X 0,Y 388.92,Z 538.848,A -85,B 0,C 180,E1 -11602.736,E2 -11602.736} C_VEL
LIN {X 0,Y 388.75,Z 543.172,A -85,B 0,C 180,E1 -11604.212,E2 -11604.212} C_VEL
LIN {X 0,Y 388.745,Z 546.747,A -85,B 0,C 180,E1 -11605.856,E2 -11605.856} C_VEL
LIN {X 0,Y 388.772,Z 548.382,A -85,B 0,C 180,E1 -11606.894,E2 -11606.894} C_VEL
LIN {X 0,Y 388.843,Z 549.555,A -85,B 0,C 180,E1 -11607.931,E2 -11607.931} C_VEL
LIN {X 0,Y 388.798,Z 550.401,A -85,B 0,C 180,E1 -11608.966,E2 -11608.966} C_VEL
LIN {X 0,Y 388.798,Z 550.686,A -85,B 0,C 180,E1 -11610.002,E2 -11610.002} C_VEL
LIN {X 0,Y 388.812,Z 550.132,A -85,B 0,C 180,E1 -11612.074,E2 -11612.074} C_VEL
LIN {X 0,Y 388.73,Z 547.698,A -85,B 0,C 180,E1 -11614.149,E2 -11614.149} C_VEL
LIN {X 0,Y 388.76,Z 545.942,A -85,B 0,C 180,E1 -11615.188,E2 -11615.188} C_VEL
LIN {X 0,Y 388.846,Z 542.291,A -85,B 0,C 180,E1 -11616.748,E2 -11616.748} C_VEL
LIN {X 0,Y 389.046,Z 537.479,A -85,B 0,C 180,E1 -11618.311,E2 -11618.311} C_VEL
LIN {X 0,Y 389.393,Z 531.34,A -85,B 0,C 180,E1 -11619.874,E2 -11619.874} C_VEL
LIN {X 0,Y 389.848,Z 525.106,A -85,B 0,C 180,E1 -11621.175,E2 -11621.175} C_VEL
LIN {X 0,Y 390.516,Z 517.594,A -85,B 0,C 180,E1 -11622.473,E2 -11622.473} C_VEL
LIN {X 0,Y 391.173,Z 508.831,A -85,B 0,C 180,E1 -11623.725,E2 -11623.725} C_VEL
LIN {X 0,Y 391.869,Z 500.869,A -85,B 0,C 180,E1 -11624.675,E2 -11624.675} C_VEL
LIN {X 0,Y 392.608,Z 491.814,A -85,B 0,C 180,E1 -11625.576,E2 -11625.576} C_VEL
LIN {X 0,Y 393.367,Z 482.401,A -85,B 0,C 180,E1 -11626.344,E2 -11626.344} C_VEL
LIN {X 0,Y 394.155,Z 471.51,A -85,B 0,C 180,E1 -11627.043,E2 -11627.043} C_VEL
LIN {X 0,Y 394.688,Z 461.213,A -85,B 0,C 180,E1 -11627.554,E2 -11627.554} C_VEL
LIN {X 0,Y 395.228,Z 450.479,A -85,B 0,C 180,E1 -11627.93,E2 -11627.93} C_VEL
LIN {X 0,Y 395.727,Z 430.363,A -85,B 0,C 180,E1 -11628.375,E2 -11628.375} C_VEL
LIN {X 0,Y 396.907,Z 367.096,A -85,B 0,C 180,E1 -11629.71,E2 -11629.71} C_VEL
LIN {X 0,Y 394.054,Z 346.926,A -85,B 0,C 180,E1 -11630.362,E2 -11630.362} C_VEL
LIN {X 0,Y 393.489,Z 343.666,A -85,B 0,C 180,E1 -11630.478,E2 -11630.478} C_VEL
LIN {X 0,Y 395.189,Z 321.392,A -85,B 0,C 180,E1 -11634.144,E2 -11634.144} C_VEL
LIN {X 0,Y 395.62,Z 314.844,A -85,B 0,C 180,E1 -11635.236,E2 -11635.236} C_VEL
LIN {X 0,Y 393.553,Z 304.918,A -85,B 0,C 180,E1 -11637.14,E2 -11637.14} C_VEL
LIN {X 0,Y 390.691,Z 294.089,A -85,B 0,C 180,E1 -11639.352,E2 -11639.352} C_VEL
LIN {X 0,Y 390.047,Z 291.906,A -85,B 0,C 180,E1 -11639.862,E2 -11639.862} C_VEL
LIN {X 0,Y 390.036,Z 291.901,A -85,B 0,C 180,E1 -11642.721,E2 -11642.721} C_VEL
LIN {X 0,Y 390.047,Z 291.904,A -85,B 0,C 180,E1 -11645.824,E2 -11645.824} C_VEL
LIN {X 0,Y 390.059,Z 291.902,A -85,B 0,C 180,E1 -11649.217,E2 -11649.217} C_VEL
LIN {X 0,Y 390.032,Z 291.904,A -85,B 0,C 180,E1 -11652.373,E2 -11652.373} C_VEL
LIN {X 0,Y 390.032,Z 291.902,A -85,B 0,C 180,E1 -11655.353,E2 -11655.353} C_VEL
LIN {X 0,Y 390.035,Z 291.9,A -85,B 0,C 180,E1 -11658.188,E2 -11658.188} C_VEL
LIN {X 0,Y 390.078,Z 291.893,A -85,B 0,C 180,E1 -11660.907,E2 -11660.907} C_VEL
LIN {X 0,Y 390.067,Z 291.889,A -85,B 0,C 180,E1 -11664.792,E2 -11664.792} C_VEL
LIN {X 0,Y 390.006,Z 291.899,A -85,B 0,C 180,E1 -11668.495,E2 -11668.495} C_VEL
LIN {X 0,Y 390.098,Z 291.886,A -85,B 0,C 180,E1 -11672.069,E2 -11672.069} C_VEL
LIN {X 0,Y 390.06,Z 291.895,A -85,B 0,C 180,E1 -11675.519,E2 -11675.519} C_VEL
LIN {X 0,Y 390.08,Z 291.895,A -85,B 0,C 180,E1 -11678.88,E2 -11678.88} C_VEL
LIN {X 0,Y 390.125,Z 291.889,A -85,B 0,C 180,E1 -11682.692,E2 -11682.692} C_VEL
LIN {X 0,Y 390.171,Z 291.884,A -85,B 0,C 180,E1 -11686.561,E2 -11686.561} C_VEL
LIN {X 0,Y 390.148,Z 291.89,A -85,B 0,C 180,E1 -11689.623,E2 -11689.623} C_VEL
LIN {X 0,Y 390.273,Z 291.878,A -85,B 0,C 180,E1 -11692.759,E2 -11692.759} C_VEL
LIN {X 0,Y 390.248,Z 292.055,A -85,B 0,C 180,E1 -11694.478,E2 -11694.478} C_VEL
LIN {X 0,Y 393.69,Z 304.596,A -85,B 0,C 180,E1 -11696.931,E2 -11696.931} C_VEL
LIN {X 0,Y 393.079,Z 320.1,A -85,B 0,C 180,E1 -11699.488,E2 -11699.488} C_VEL
LIN {X 0,Y 392.447,Z 338.222,A -85,B 0,C 180,E1 -11702.457,E2 -11702.457} C_VEL
LIN {X 0,Y 396.349,Z 359.585,A -85,B 0,C 180,E1 -11703.281,E2 -11703.281} C_VEL
LIN {X 0,Y 396.42,Z 365.853,A -85,B 0,C 180,E1 -11703.449,E2 -11703.449} C_VEL
LIN {X 0,Y 394.795,Z 424.233,A -85,B 0,C 180,E1 -11704.887,E2 -11704.887} C_VEL
LIN {X 0,Y 394.344,Z 435.094,A -85,B 0,C 180,E1 -11705.305,E2 -11705.305} C_VEL
LIN {X 0,Y 393.744,Z 447.475,A -85,B 0,C 180,E1 -11706.02,E2 -11706.02} C_VEL
LIN {X 0,Y 393.273,Z 455.998,A -85,B 0,C 180,E1 -11706.671,E2 -11706.671} C_VEL
LIN {X 0,Y 392.661,Z 464.367,A -85,B 0,C 180,E1 -11707.456,E2 -11707.456} C_VEL
LIN {X 0,Y 392.082,Z 471.353,A -85,B 0,C 180,E1 -11708.245,E2 -11708.245} C_VEL
LIN {X 0,Y 391.502,Z 478.105,A -85,B 0,C 180,E1 -11709.155,E2 -11709.155} C_VEL
LIN {X 0,Y 391.001,Z 483.968,A -85,B 0,C 180,E1 -11710.094,E2 -11710.094} C_VEL
LIN {X 0,Y 390.521,Z 489.514,A -85,B 0,C 180,E1 -11711.155,E2 -11711.155} C_VEL
LIN {X 0,Y 390.089,Z 494.159,A -85,B 0,C 180,E1 -11712.222,E2 -11712.222} C_VEL
LIN {X 0,Y 389.667,Z 498.809,A -85,B 0,C 180,E1 -11713.561,E2 -11713.561} C_VEL
LIN {X 0,Y 389.277,Z 503.01,A -85,B 0,C 180,E1 -11715.176,E2 -11715.176} C_VEL
LIN {X 0,Y 389.178,Z 504.166,A -85,B 0,C 180,E1 -11715.717,E2 -11715.717} C_VEL
LIN {X 0,Y 389.001,Z 505.862,A -85,B 0,C 180,E1 -11716.803,E2 -11716.803} C_VEL
LIN {X 0,Y 388.817,Z 506.952,A -85,B 0,C 180,E1 -11717.896,E2 -11717.896} C_VEL
LIN {X 0,Y 388.72,Z 507.486,A -85,B 0,C 180,E1 -11718.993,E2 -11718.993} C_VEL
LIN {X 0,Y 388.687,Z 507.467,A -85,B 0,C 180,E1 -11720.094,E2 -11720.094} C_VEL
LIN {X 0,Y 388.704,Z 506.883,A -85,B 0,C 180,E1 -11721.2,E2 -11721.2} C_VEL
LIN {X 0,Y 388.845,Z 504.852,A -85,B 0,C 180,E1 -11722.821,E2 -11722.821} C_VEL
LIN {X 0,Y 388.987,Z 502.612,A -85,B 0,C 180,E1 -11723.987,E2 -11723.987} C_VEL
LIN {X 0,Y 389.195,Z 498.662,A -85,B 0,C 180,E1 -11725.467,E2 -11725.467} C_VEL
LIN {X 0,Y 389.423,Z 493.902,A -85,B 0,C 180,E1 -11726.82,E2 -11726.82} C_VEL
LIN {X 0,Y 389.787,Z 487.506,A -85,B 0,C 180,E1 -11728.249,E2 -11728.249} C_VEL
LIN {X 0,Y 390.294,Z 479.152,A -85,B 0,C 180,E1 -11729.683,E2 -11729.683} C_VEL
LIN {X 0,Y 390.701,Z 471.855,A -85,B 0,C 180,E1 -11730.692,E2 -11730.692} C_VEL
LIN {X 0,Y 391.149,Z 464.326,A -85,B 0,C 180,E1 -11731.555,E2 -11731.555} C_VEL
LIN {X 0,Y 391.578,Z 456.793,A -85,B 0,C 180,E1 -11732.273,E2 -11732.273} C_VEL
LIN {X 0,Y 391.936,Z 448.485,A -85,B 0,C 180,E1 -11732.926,E2 -11732.926} C_VEL
LIN {X 0,Y 392.328,Z 439.221,A -85,B 0,C 180,E1 -11733.502,E2 -11733.502} C_VEL
LIN {X 0,Y 392.613,Z 429.106,A -85,B 0,C 180,E1 -11733.976,E2 -11733.976} C_VEL
LIN {X 0,Y 392.873,Z 417.635,A -85,B 0,C 180,E1 -11734.337,E2 -11734.337} C_VEL
LIN {X 0,Y 393.862,Z 359.667,A -85,B 0,C 180,E1 -11735.622,E2 -11735.622} C_VEL
LIN {X 0,Y 390.947,Z 339.387,A -85,B 0,C 180,E1 -11736.203,E2 -11736.203} C_VEL
LIN {X 0,Y 391.738,Z 325.371,A -85,B 0,C 180,E1 -11739.214,E2 -11739.214} C_VEL
LIN {X 0,Y 392.712,Z 308.81,A -85,B 0,C 180,E1 -11742.848,E2 -11742.848} C_VEL
LIN {X 0,Y 392.491,Z 304.217,A -85,B 0,C 180,E1 -11743.9,E2 -11743.9} C_VEL
LIN {X 0,Y 390.089,Z 291.894,A -85,B 0,C 180,E1 -11746.913,E2 -11746.913} C_VEL
LIN {X 0,Y 390.053,Z 291.895,A -85,B 0,C 180,E1 -11750.905,E2 -11750.905} C_VEL
LIN {X 0,Y 390.066,Z 291.892,A -85,B 0,C 180,E1 -11754.793,E2 -11754.793} C_VEL
LIN {X 0,Y 390.02,Z 291.899,A -85,B 0,C 180,E1 -11758.496,E2 -11758.496} C_VEL
LIN {X 0,Y 390.016,Z 291.904,A -85,B 0,C 180,E1 -11762.004,E2 -11762.004} C_VEL
LIN {X 0,Y 390.043,Z 291.895,A -85,B 0,C 180,E1 -11765.517,E2 -11765.517} C_VEL
LIN {X 0,Y 390.055,Z 291.896,A -85,B 0,C 180,E1 -11768.878,E2 -11768.878} C_VEL
LIN {X 0,Y 390.115,Z 291.887,A -85,B 0,C 180,E1 -11772.166,E2 -11772.166} C_VEL
LIN {X 0,Y 390.142,Z 291.884,A -85,B 0,C 180,E1 -11775.392,E2 -11775.392} C_VEL
LIN {X 0,Y 390.148,Z 291.884,A -85,B 0,C 180,E1 -11778.57,E2 -11778.57} C_VEL
LIN {X 0,Y 390.262,Z 291.868,A -85,B 0,C 180,E1 -11782.085,E2 -11782.085} C_VEL
LIN {X 0,Y 390.202,Z 291.876,A -85,B 0,C 180,E1 -11784.832,E2 -11784.832} C_VEL
LIN {X 0,Y 390.359,Z 291.856,A -85,B 0,C 180,E1 -11788.251,E2 -11788.251} C_VEL
LIN {X 0,Y 390.407,Z 291.854,A -85,B 0,C 180,E1 -11792.061,E2 -11792.061} C_VEL
LIN {X 0,Y 390.279,Z 291.865,A -85,B 0,C 180,E1 -11792.751,E2 -11792.751} C_VEL
LIN {X 0,Y 389.531,Z 291.964,A -85,B 0,C 180,E1 -11793.612,E2 -11793.612} C_VEL
LIN {X 0,Y 386.65,Z 292.317,A -85,B 0,C 180,E1 -11795.011,E2 -11795.011} C_VEL
LIN {X 0,Y 384.272,Z 292.621,A -85,B 0,C 180,E1 -11796.142,E2 -11796.142} C_VEL
LIN {X 0,Y 383.272,Z 292.739,A -85,B 0,C 180,E1 -11797.016,E2 -11797.016} C_VEL
LIN {X 0,Y 383.199,Z 292.747,A -85,B 0,C 180,E1 -11797.312,E2 -11797.312} C_VEL
LIN {X 0,Y 383.125,Z 292.761,A -85,B 0,C 180,E1 -11800.567,E2 -11800.567} C_VEL
LIN {X 0,Y 383.125,Z 292.757,A -85,B 0,C 180,E1 -11803.793,E2 -11803.793} C_VEL
LIN {X 0,Y 383.072,Z 292.764,A -85,B 0,C 180,E1 -11807.441,E2 -11807.441} C_VEL
LIN {X 0,Y 383.023,Z 292.773,A -85,B 0,C 180,E1 -11810.643,E2 -11810.643} C_VEL
LIN {X 0,Y 383.004,Z 292.772,A -85,B 0,C 180,E1 -11813.804,E2 -11813.804} C_VEL
LIN {X 0,Y 382.976,Z 292.783,A -85,B 0,C 180,E1 -11817.303,E2 -11817.303} C_VEL
LIN {X 0,Y 382.967,Z 292.777,A -85,B 0,C 180,E1 -11820.914,E2 -11820.914} C_VEL
LIN {X 0,Y 383,Z 292.772,A -85,B 0,C 180,E1 -11824.663,E2 -11824.663} C_VEL
LIN {X 0,Y 382.976,Z 292.783,A -85,B 0,C 180,E1 -11827.898,E2 -11827.898} C_VEL
LIN {X 0,Y 382.946,Z 292.779,A -85,B 0,C 180,E1 -11831.344,E2 -11831.344} C_VEL
LIN {X 0,Y 382.968,Z 292.784,A -85,B 0,C 180,E1 -11834.298,E2 -11834.298} C_VEL
LIN {X 0,Y 382.982,Z 292.775,A -85,B 0,C 180,E1 -11837.235,E2 -11837.235} C_VEL
LIN {X 0,Y 382.982,Z 292.779,A -85,B 0,C 180,E1 -11840.409,E2 -11840.409} C_VEL
LIN {X 0,Y 382.978,Z 292.775,A -85,B 0,C 180,E1 -11844.039,E2 -11844.039} C_VEL
LIN {X 0,Y 382.946,Z 292.78,A -85,B 0,C 180,E1 -11847.575,E2 -11847.575} C_VEL
LIN {X 0,Y 382.956,Z 292.778,A -85,B 0,C 180,E1 -11850.296,E2 -11850.296} C_VEL
LIN {X 0,Y 383.015,Z 292.771,A -85,B 0,C 180,E1 -11852.694,E2 -11852.694} C_VEL
LIN {X 0,Y 383.006,Z 292.774,A -85,B 0,C 180,E1 -11855.036,E2 -11855.036} C_VEL
LIN {X 0,Y 382.944,Z 292.779,A -85,B 0,C 180,E1 -11858.466,E2 -11858.466} C_VEL
LIN {X 0,Y 383.004,Z 292.779,A -85,B 0,C 180,E1 -11861.823,E2 -11861.823} C_VEL
LIN {X 0,Y 383.061,Z 292.764,A -85,B 0,C 180,E1 -11865.116,E2 -11865.116} C_VEL
LIN {X 0,Y 383.054,Z 292.771,A -85,B 0,C 180,E1 -11868.356,E2 -11868.356} C_VEL
LIN {X 0,Y 383.213,Z 292.748,A -85,B 0,C 180,E1 -11871.974,E2 -11871.974} C_VEL
LIN {X 0,Y 383.148,Z 292.759,A -85,B 0,C 180,E1 -11874.737,E2 -11874.737} C_VEL
LIN {X 0,Y 383.336,Z 292.73,A -85,B 0,C 180,E1 -11877.898,E2 -11877.898} C_VEL
LIN {X 0,Y 383.464,Z 292.714,A -85,B 0,C 180,E1 -11879.999,E2 -11879.999} C_VEL
LIN {X 0,Y 383.203,Z 292.754,A -85,B 0,C 180,E1 -11883.153,E2 -11883.153} C_VEL
LIN {X 0,Y 383.23,Z 292.743,A -85,B 0,C 180,E1 -11886.317,E2 -11886.317} C_VEL
LIN {X 0,Y 383.17,Z 292.751,A -85,B 0,C 180,E1 -11888.437,E2 -11888.437} C_VEL
LIN {X 0,Y 383.053,Z 292.772,A -85,B 0,C 180,E1 -11891.643,E2 -11891.643} C_VEL
LIN {X 0,Y 383.059,Z 292.765,A -85,B 0,C 180,E1 -11894.883,E2 -11894.883} C_VEL
LIN {X 0,Y 383.011,Z 292.775,A -85,B 0,C 180,E1 -11898.175,E2 -11898.175} C_VEL
LIN {X 0,Y 382.945,Z 292.78,A -85,B 0,C 180,E1 -11901.533,E2 -11901.533} C_VEL
LIN {X 0,Y 383.005,Z 292.772,A -85,B 0,C 180,E1 -11904.963,E2 -11904.963} C_VEL
LIN {X 0,Y 382.982,Z 292.779,A -85,B 0,C 180,E1 -11908.272,E2 -11908.272} C_VEL
LIN {X 0,Y 382.964,Z 292.778,A -85,B 0,C 180,E1 -11912.153,E2 -11912.153} C_VEL
LIN {X 0,Y 382.977,Z 292.78,A -85,B 0,C 180,E1 -11914.671,E2 -11914.671} C_VEL
LIN {X 0,Y 382.959,Z 292.777,A -85,B 0,C 180,E1 -11917.907,E2 -11917.907} C_VEL
LIN {X 0,Y 382.942,Z 292.786,A -85,B 0,C 180,E1 -11921.352,E2 -11921.352} C_VEL
LIN {X 0,Y 382.96,Z 292.777,A -85,B 0,C 180,E1 -11924.307,E2 -11924.307} C_VEL
LIN {X 0,Y 382.98,Z 292.778,A -85,B 0,C 180,E1 -11927.244,E2 -11927.244} C_VEL
LIN {X 0,Y 382.969,Z 292.777,A -85,B 0,C 180,E1 -11930.421,E2 -11930.421} C_VEL
LIN {X 0,Y 382.987,Z 292.781,A -85,B 0,C 180,E1 -11934.047,E2 -11934.047} C_VEL
LIN {X 0,Y 382.962,Z 292.778,A -85,B 0,C 180,E1 -11937.583,E2 -11937.583} C_VEL
LIN {X 0,Y 383.043,Z 292.915,A -85,B 0,C 180,E1 -11940.613,E2 -11940.613} C_VEL
LIN {X 0,Y 386.539,Z 308.972,A -85,B 0,C 180,E1 -11943.888,E2 -11943.888} C_VEL
LIN {X 0,Y 387.724,Z 314.579,A -85,B 0,C 180,E1 -11945,E2 -11945} C_VEL
LIN {X 0,Y 386.42,Z 330.716,A -85,B 0,C 180,E1 -11947.905,E2 -11947.905} C_VEL
LIN {X 0,Y 385.273,Z 344.485,A -85,B 0,C 180,E1 -11950.36,E2 -11950.36} C_VEL
LIN {X 0,Y 388.048,Z 369.474,A -85,B 0,C 180,E1 -11951.02,E2 -11951.02} C_VEL
LIN {X 0,Y 386.716,Z 449.588,A -85,B 0,C 180,E1 -11952.691,E2 -11952.691} C_VEL
LIN {X 0,Y 386.329,Z 459.383,A -85,B 0,C 180,E1 -11953.014,E2 -11953.014} C_VEL
LIN {X 0,Y 385.88,Z 469.28,A -85,B 0,C 180,E1 -11953.47,E2 -11953.47} C_VEL
LIN {X 0,Y 385.437,Z 478.12,A -85,B 0,C 180,E1 -11953.995,E2 -11953.995} C_VEL
LIN {X 0,Y 384.795,Z 488.577,A -85,B 0,C 180,E1 -11954.782,E2 -11954.782} C_VEL
LIN {X 0,Y 384.3,Z 496.982,A -85,B 0,C 180,E1 -11955.556,E2 -11955.556} C_VEL
LIN {X 0,Y 383.742,Z 505.525,A -85,B 0,C 180,E1 -11956.5,E2 -11956.5} C_VEL
LIN {X 0,Y 383.161,Z 513.536,A -85,B 0,C 180,E1 -11957.557,E2 -11957.557} C_VEL
LIN {X 0,Y 382.622,Z 521.807,A -85,B 0,C 180,E1 -11958.883,E2 -11958.883} C_VEL
LIN {X 0,Y 382.239,Z 528.649,A -85,B 0,C 180,E1 -11960.211,E2 -11960.211} C_VEL
LIN {X 0,Y 381.984,Z 534.319,A -85,B 0,C 180,E1 -11961.539,E2 -11961.539} C_VEL
LIN {X 0,Y 381.843,Z 538.191,A -85,B 0,C 180,E1 -11962.6,E2 -11962.6} C_VEL
LIN {X 0,Y 381.659,Z 542.936,A -85,B 0,C 180,E1 -11964.254,E2 -11964.254} C_VEL
LIN {X 0,Y 381.677,Z 546.227,A -85,B 0,C 180,E1 -11965.779,E2 -11965.779} C_VEL
LIN {X 0,Y 381.679,Z 547.863,A -85,B 0,C 180,E1 -11966.836,E2 -11966.836} C_VEL
LIN {X 0,Y 381.775,Z 549.085,A -85,B 0,C 180,E1 -11967.892,E2 -11967.892} C_VEL
LIN {X 0,Y 381.728,Z 549.968,A -85,B 0,C 180,E1 -11968.947,E2 -11968.947} C_VEL
LIN {X 0,Y 381.717,Z 550.179,A -85,B 0,C 180,E1 -11971.057,E2 -11971.057} C_VEL
LIN {X 0,Y 381.725,Z 549.762,A -85,B 0,C 180,E1 -11972.112,E2 -11972.112} C_VEL
LIN {X 0,Y 381.653,Z 547.375,A -85,B 0,C 180,E1 -11974.226,E2 -11974.226} C_VEL
LIN {X 0,Y 381.657,Z 545.627,A -85,B 0,C 180,E1 -11975.284,E2 -11975.284} C_VEL
LIN {X 0,Y 381.778,Z 542.007,A -85,B 0,C 180,E1 -11976.874,E2 -11976.874} C_VEL
LIN {X 0,Y 381.983,Z 537.244,A -85,B 0,C 180,E1 -11978.465,E2 -11978.465} C_VEL
LIN {X 0,Y 382.371,Z 531.169,A -85,B 0,C 180,E1 -11980.057,E2 -11980.057} C_VEL
LIN {X 0,Y 382.863,Z 525.002,A -85,B 0,C 180,E1 -11981.382,E2 -11981.382} C_VEL
LIN {X 0,Y 383.555,Z 517.545,A -85,B 0,C 180,E1 -11982.703,E2 -11982.703} C_VEL
LIN {X 0,Y 384.227,Z 509.175,A -85,B 0,C 180,E1 -11983.933,E2 -11983.933} C_VEL
LIN {X 0,Y 385.103,Z 499.703,A -85,B 0,C 180,E1 -11985.074,E2 -11985.074} C_VEL
LIN {X 0,Y 385.909,Z 490.467,A -85,B 0,C 180,E1 -11985.989,E2 -11985.989} C_VEL
LIN {X 0,Y 386.721,Z 480.81,A -85,B 0,C 180,E1 -11986.769,E2 -11986.769} C_VEL
LIN {X 0,Y 387.458,Z 470.76,A -85,B 0,C 180,E1 -11987.415,E2 -11987.415} C_VEL
LIN {X 0,Y 388.04,Z 460.393,A -85,B 0,C 180,E1 -11987.933,E2 -11987.933} C_VEL
LIN {X 0,Y 388.569,Z 449.542,A -85,B 0,C 180,E1 -11988.316,E2 -11988.316} C_VEL
LIN {X 0,Y 389.216,Z 421.796,A -85,B 0,C 180,E1 -11988.933,E2 -11988.933} C_VEL
LIN {X 0,Y 390.34,Z 367.454,A -85,B 0,C 180,E1 -11990.117,E2 -11990.117} C_VEL
LIN {X 0,Y 387.5,Z 347.604,A -85,B 0,C 180,E1 -11990.78,E2 -11990.78} C_VEL
LIN {X 0,Y 386.806,Z 343.4,A -85,B 0,C 180,E1 -11990.963,E2 -11990.963} C_VEL
LIN {X 0,Y 388.714,Z 320.174,A -85,B 0,C 180,E1 -11994.858,E2 -11994.858} C_VEL
LIN {X 0,Y 388.941,Z 317.074,A -85,B 0,C 180,E1 -11995.382,E2 -11995.382} C_VEL
LIN {X 0,Y 386.995,Z 307.383,A -85,B 0,C 180,E1 -11997.292,E2 -11997.292} C_VEL
LIN {X 0,Y 383.689,Z 295.118,A -85,B 0,C 180,E1 -11999.875,E2 -11999.875} C_VEL
LIN {X 0,Y 382.99,Z 292.784,A -85,B 0,C 180,E1 -12000.406,E2 -12000.406} C_VEL
LIN {X 0,Y 382.996,Z 292.78,A -85,B 0,C 180,E1 -12003.4,E2 -12003.4} C_VEL
LIN {X 0,Y 383.023,Z 292.776,A -85,B 0,C 180,E1 -12006.164,E2 -12006.164} C_VEL
LIN {X 0,Y 382.998,Z 292.78,A -85,B 0,C 180,E1 -12009.958,E2 -12009.958} C_VEL
LIN {X 0,Y 382.995,Z 292.779,A -85,B 0,C 180,E1 -12012.778,E2 -12012.778} C_VEL
LIN {X 0,Y 382.985,Z 292.778,A -85,B 0,C 180,E1 -12015.788,E2 -12015.788} C_VEL
LIN {X 0,Y 382.992,Z 292.777,A -85,B 0,C 180,E1 -12018.792,E2 -12018.792} C_VEL
LIN {X 0,Y 382.987,Z 292.775,A -85,B 0,C 180,E1 -12022.095,E2 -12022.095} C_VEL
LIN {X 0,Y 383.001,Z 292.769,A -85,B 0,C 180,E1 -12025.331,E2 -12025.331} C_VEL
LIN {X 0,Y 382.966,Z 292.772,A -85,B 0,C 180,E1 -12029.081,E2 -12029.081} C_VEL
LIN {X 0,Y 383.037,Z 292.771,A -85,B 0,C 180,E1 -12032.697,E2 -12032.697} C_VEL
LIN {X 0,Y 383.022,Z 292.772,A -85,B 0,C 180,E1 -12036.193,E2 -12036.193} C_VEL
LIN {X 0,Y 383.059,Z 292.769,A -85,B 0,C 180,E1 -12039.599,E2 -12039.599} C_VEL
LIN {X 0,Y 383.081,Z 292.767,A -85,B 0,C 180,E1 -12042.931,E2 -12042.931} C_VEL
LIN {X 0,Y 383.103,Z 292.764,A -85,B 0,C 180,E1 -12046.464,E2 -12046.464} C_VEL
LIN {X 0,Y 383.112,Z 292.767,A -85,B 0,C 180,E1 -12049.43,E2 -12049.43} C_VEL
LIN {X 0,Y 383.225,Z 292.756,A -85,B 0,C 180,E1 -12052.625,E2 -12052.625} C_VEL
LIN {X 0,Y 383.26,Z 292.822,A -85,B 0,C 180,E1 -12053.915,E2 -12053.915} C_VEL
LIN {X 0,Y 387.131,Z 307.606,A -85,B 0,C 180,E1 -12056.879,E2 -12056.879} C_VEL
LIN {X 0,Y 386.116,Z 329.383,A -85,B 0,C 180,E1 -12060.522,E2 -12060.522} C_VEL
LIN {X 0,Y 385.729,Z 338.241,A -85,B 0,C 180,E1 -12061.991,E2 -12061.991} C_VEL
LIN {X 0,Y 389.257,Z 356.91,A -85,B 0,C 180,E1 -12062.749,E2 -12062.749} C_VEL
LIN {X 0,Y 390.011,Z 363.102,A -85,B 0,C 180,E1 -12062.966,E2 -12062.966} C_VEL
LIN {X 0,Y 388.16,Z 424.527,A -85,B 0,C 180,E1 -12064.521,E2 -12064.521} C_VEL
LIN {X 0,Y 387.652,Z 436.696,A -85,B 0,C 180,E1 -12065.011,E2 -12065.011} C_VEL
LIN {X 0,Y 386.981,Z 448.51,A -85,B 0,C 180,E1 -12065.733,E2 -12065.733} C_VEL
LIN {X 0,Y 386.506,Z 456.849,A -85,B 0,C 180,E1 -12066.395,E2 -12066.395} C_VEL
LIN {X 0,Y 385.901,Z 463.931,A -85,B 0,C 180,E1 -12067.062,E2 -12067.062} C_VEL
LIN {X 0,Y 385.235,Z 472.075,A -85,B 0,C 180,E1 -12067.997,E2 -12067.997} C_VEL
LIN {X 0,Y 384.563,Z 479.3,A -85,B 0,C 180,E1 -12069.002,E2 -12069.002} C_VEL
LIN {X 0,Y 384.019,Z 485.337,A -85,B 0,C 180,E1 -12070.013,E2 -12070.013} C_VEL
LIN {X 0,Y 383.509,Z 490.729,A -85,B 0,C 180,E1 -12071.095,E2 -12071.095} C_VEL
LIN {X 0,Y 383.049,Z 495.236,A -85,B 0,C 180,E1 -12072.181,E2 -12072.181} C_VEL
LIN {X 0,Y 382.683,Z 498.969,A -85,B 0,C 180,E1 -12073.273,E2 -12073.273} C_VEL
LIN {X 0,Y 382.411,Z 502.013,A -85,B 0,C 180,E1 -12074.366,E2 -12074.366} C_VEL
LIN {X 0,Y 382.155,Z 504.406,A -85,B 0,C 180,E1 -12075.466,E2 -12075.466} C_VEL
LIN {X 0,Y 381.879,Z 506.786,A -85,B 0,C 180,E1 -12077.126,E2 -12077.126} C_VEL
LIN {X 0,Y 381.696,Z 507.723,A -85,B 0,C 180,E1 -12078.242,E2 -12078.242} C_VEL
LIN {X 0,Y 381.639,Z 508.005,A -85,B 0,C 180,E1 -12079.359,E2 -12079.359} C_VEL
LIN {X 0,Y 381.6,Z 507.695,A -85,B 0,C 180,E1 -12080.483,E2 -12080.483} C_VEL
LIN {X 0,Y 381.625,Z 506.819,A -85,B 0,C 180,E1 -12081.613,E2 -12081.613} C_VEL
LIN {X 0,Y 381.793,Z 504.884,A -85,B 0,C 180,E1 -12083.024,E2 -12083.024} C_VEL
LIN {X 0,Y 381.958,Z 501.915,A -85,B 0,C 180,E1 -12084.457,E2 -12084.457} C_VEL
LIN {X 0,Y 382.133,Z 498.452,A -85,B 0,C 180,E1 -12085.693,E2 -12085.693} C_VEL
LIN {X 0,Y 382.402,Z 493.582,A -85,B 0,C 180,E1 -12087.057,E2 -12087.057} C_VEL
LIN {X 0,Y 382.802,Z 486.972,A -85,B 0,C 180,E1 -12088.513,E2 -12088.513} C_VEL
LIN {X 0,Y 383.204,Z 480.244,A -85,B 0,C 180,E1 -12089.682,E2 -12089.682} C_VEL
LIN {X 0,Y 383.689,Z 471.915,A -85,B 0,C 180,E1 -12090.856,E2 -12090.856} C_VEL
LIN {X 0,Y 384.138,Z 464.313,A -85,B 0,C 180,E1 -12091.736,E2 -12091.736} C_VEL
LIN {X 0,Y 384.627,Z 455.888,A -85,B 0,C 180,E1 -12092.538,E2 -12092.538} C_VEL
LIN {X 0,Y 385.037,Z 447.29,A -85,B 0,C 180,E1 -12093.202,E2 -12093.202} C_VEL
LIN {X 0,Y 385.469,Z 436.279,A -85,B 0,C 180,E1 -12093.865,E2 -12093.865} C_VEL
LIN {X 0,Y 385.819,Z 424.701,A -85,B 0,C 180,E1 -12094.342,E2 -12094.342} C_VEL
LIN {X 0,Y 386.23,Z 403.68,A -85,B 0,C 180,E1 -12094.855,E2 -12094.855} C_VEL
LIN {X 0,Y 386.983,Z 360.804,A -85,B 0,C 180,E1 -12095.832,E2 -12095.832} C_VEL
LIN {X 0,Y 383.954,Z 339.411,A -85,B 0,C 180,E1 -12096.467,E2 -12096.467} C_VEL
LIN {X 0,Y 384.896,Z 323.575,A -85,B 0,C 180,E1 -12099.927,E2 -12099.927} C_VEL
LIN {X 0,Y 385.805,Z 308.766,A -85,B 0,C 180,E1 -12103.229,E2 -12103.229} C_VEL
LIN {X 0,Y 385.326,Z 304.583,A -85,B 0,C 180,E1 -12104.222,E2 -12104.222} C_VEL
LIN {X 0,Y 383.034,Z 292.772,A -85,B 0,C 180,E1 -12107.166,E2 -12107.166} C_VEL
LIN {X 0,Y 382.982,Z 292.776,A -85,B 0,C 180,E1 -12110.421,E2 -12110.421} C_VEL
LIN {X 0,Y 383.01,Z 292.774,A -85,B 0,C 180,E1 -12114.044,E2 -12114.044} C_VEL
LIN {X 0,Y 382.984,Z 292.778,A -85,B 0,C 180,E1 -12117.58,E2 -12117.58} C_VEL
LIN {X 0,Y 382.975,Z 292.779,A -85,B 0,C 180,E1 -12120.3,E2 -12120.3} C_VEL
LIN {X 0,Y 383.004,Z 292.777,A -85,B 0,C 180,E1 -12124.046,E2 -12124.046} C_VEL
LIN {X 0,Y 382.988,Z 292.774,A -85,B 0,C 180,E1 -12127.334,E2 -12127.334} C_VEL
LIN {X 0,Y 383.053,Z 292.772,A -85,B 0,C 180,E1 -12130.716,E2 -12130.716} C_VEL
LIN {X 0,Y 383.081,Z 292.762,A -85,B 0,C 180,E1 -12134.026,E2 -12134.026} C_VEL
LIN {X 0,Y 383.141,Z 292.759,A -85,B 0,C 180,E1 -12137.283,E2 -12137.283} C_VEL
LIN {X 0,Y 383.143,Z 292.755,A -85,B 0,C 180,E1 -12140.497,E2 -12140.497} C_VEL
LIN {X 0,Y 383.238,Z 292.746,A -85,B 0,C 180,E1 -12143.681,E2 -12143.681} C_VEL
LIN {X 0,Y 383.372,Z 292.73,A -85,B 0,C 180,E1 -12147.897,E2 -12147.897} C_VEL
LIN {X 0,Y 383.372,Z 292.73,A -85,B 0,C 180,E1 -12152.099,E2 -12152.099} C_VEL
LIN {X 0,Y 383.235,Z 292.748,A -85,B 0,C 180,E1 -12156.314,E2 -12156.314} C_VEL
LIN {X 0,Y 383.199,Z 292.747,A -85,B 0,C 180,E1 -12157.312,E2 -12157.312} C_VEL
LIN {X 0,Y 382.54,Z 292.837,A -85,B 0,C 180,E1 -12158.189,E2 -12158.189} C_VEL
LIN {X 0,Y 379.643,Z 293.197,A -85,B 0,C 180,E1 -12159.612,E2 -12159.612} C_VEL
LIN {X 0,Y 377.181,Z 293.503,A -85,B 0,C 180,E1 -12160.763,E2 -12160.763} C_VEL
LIN {X 0,Y 376.128,Z 293.631,A -85,B 0,C 180,E1 -12161.655,E2 -12161.655} C_VEL
LIN {X 0,Y 376.045,Z 293.639,A -85,B 0,C 180,E1 -12161.957,E2 -12161.957} C_VEL
LIN {X 0,Y 376.055,Z 293.639,A -85,B 0,C 180,E1 -12165.164,E2 -12165.164} C_VEL
LIN {X 0,Y 375.998,Z 293.648,A -85,B 0,C 180,E1 -12168.523,E2 -12168.523} C_VEL
LIN {X 0,Y 375.949,Z 293.65,A -85,B 0,C 180,E1 -12171.95,E2 -12171.95} C_VEL
LIN {X 0,Y 375.941,Z 293.656,A -85,B 0,C 180,E1 -12175.461,E2 -12175.461} C_VEL
LIN {X 0,Y 375.905,Z 293.66,A -85,B 0,C 180,E1 -12179.079,E2 -12179.079} C_VEL
LIN {X 0,Y 375.942,Z 293.659,A -85,B 0,C 180,E1 -12181.557,E2 -12181.557} C_VEL
LIN {X 0,Y 375.939,Z 293.655,A -85,B 0,C 180,E1 -12185.411,E2 -12185.411} C_VEL
LIN {X 0,Y 375.95,Z 293.654,A -85,B 0,C 180,E1 -12188.265,E2 -12188.265} C_VEL
LIN {X 0,Y 375.9,Z 293.658,A -85,B 0,C 180,E1 -12191.594,E2 -12191.594} C_VEL
LIN {X 0,Y 375.898,Z 293.657,A -85,B 0,C 180,E1 -12195.264,E2 -12195.264} C_VEL
LIN {X 0,Y 375.904,Z 293.662,A -85,B 0,C 180,E1 -12198.395,E2 -12198.395} C_VEL
LIN {X 0,Y 375.939,Z 293.652,A -85,B 0,C 180,E1 -12201.726,E2 -12201.726} C_VEL
LIN {X 0,Y 375.938,Z 293.654,A -85,B 0,C 180,E1 -12205.33,E2 -12205.33} C_VEL
LIN {X 0,Y 375.918,Z 293.655,A -85,B 0,C 180,E1 -12208.434,E2 -12208.434} C_VEL
LIN {X 0,Y 375.955,Z 293.65,A -85,B 0,C 180,E1 -12212.137,E2 -12212.137} C_VEL
LIN {X 0,Y 375.962,Z 293.649,A -85,B 0,C 180,E1 -12214.535,E2 -12214.535} C_VEL
LIN {X 0,Y 375.909,Z 293.658,A -85,B 0,C 180,E1 -12218.042,E2 -12218.042} C_VEL
LIN {X 0,Y 375.952,Z 293.653,A -85,B 0,C 180,E1 -12221.47,E2 -12221.47} C_VEL
LIN {X 0,Y 376.009,Z 293.643,A -85,B 0,C 180,E1 -12224.83,E2 -12224.83} C_VEL
LIN {X 0,Y 376.006,Z 293.65,A -85,B 0,C 180,E1 -12228.135,E2 -12228.135} C_VEL
LIN {X 0,Y 376.169,Z 293.625,A -85,B 0,C 180,E1 -12231.917,E2 -12231.917} C_VEL
LIN {X 0,Y 376.12,Z 293.636,A -85,B 0,C 180,E1 -12234.639,E2 -12234.639} C_VEL
LIN {X 0,Y 376.304,Z 293.606,A -85,B 0,C 180,E1 -12237.859,E2 -12237.859} C_VEL
LIN {X 0,Y 376.434,Z 293.59,A -85,B 0,C 180,E1 -12239.999,E2 -12239.999} C_VEL
LIN {X 0,Y 376.141,Z 293.632,A -85,B 0,C 180,E1 -12243.213,E2 -12243.213} C_VEL
LIN {X 0,Y 376.188,Z 293.621,A -85,B 0,C 180,E1 -12246.435,E2 -12246.435} C_VEL
LIN {X 0,Y 376.067,Z 293.64,A -85,B 0,C 180,E1 -12249.682,E2 -12249.682} C_VEL
LIN {X 0,Y 376.039,Z 293.647,A -85,B 0,C 180,E1 -12253.659,E2 -12253.659} C_VEL
LIN {X 0,Y 375.993,Z 293.649,A -85,B 0,C 180,E1 -12257.607,E2 -12257.607} C_VEL
LIN {X 0,Y 375.931,Z 293.653,A -85,B 0,C 180,E1 -12260.834,E2 -12260.834} C_VEL
LIN {X 0,Y 375.947,Z 293.659,A -85,B 0,C 180,E1 -12264.284,E2 -12264.284} C_VEL
LIN {X 0,Y 375.974,Z 293.652,A -85,B 0,C 180,E1 -12266.655,E2 -12266.655} C_VEL
LIN {X 0,Y 375.919,Z 293.658,A -85,B 0,C 180,E1 -12270.316,E2 -12270.316} C_VEL
LIN {X 0,Y 375.919,Z 293.655,A -85,B 0,C 180,E1 -12274.115,E2 -12274.115} C_VEL
LIN {X 0,Y 375.913,Z 293.659,A -85,B 0,C 180,E1 -12276.745,E2 -12276.745} C_VEL
LIN {X 0,Y 375.939,Z 293.652,A -85,B 0,C 180,E1 -12279.972,E2 -12279.972} C_VEL
LIN {X 0,Y 375.895,Z 293.66,A -85,B 0,C 180,E1 -12283.77,E2 -12283.77} C_VEL
LIN {X 0,Y 375.903,Z 293.657,A -85,B 0,C 180,E1 -12286.815,E2 -12286.815} C_VEL
LIN {X 0,Y 375.917,Z 293.655,A -85,B 0,C 180,E1 -12290.539,E2 -12290.539} C_VEL
LIN {X 0,Y 375.931,Z 293.655,A -85,B 0,C 180,E1 -12293.501,E2 -12293.501} C_VEL
LIN {X 0,Y 375.934,Z 293.657,A -85,B 0,C 180,E1 -12295.892,E2 -12295.892} C_VEL
LIN {X 0,Y 375.945,Z 293.653,A -85,B 0,C 180,E1 -12299.691,E2 -12299.691} C_VEL
LIN {X 0,Y 375.993,Z 293.816,A -85,B 0,C 180,E1 -12300.314,E2 -12300.314} C_VEL
LIN {X 0,Y 379.52,Z 309.645,A -85,B 0,C 180,E1 -12303.618,E2 -12303.618} C_VEL
LIN {X 0,Y 380.799,Z 315.948,A -85,B 0,C 180,E1 -12304.887,E2 -12304.887} C_VEL
LIN {X 0,Y 379.343,Z 332.968,A -85,B 0,C 180,E1 -12308.006,E2 -12308.006} C_VEL
LIN {X 0,Y 378.331,Z 344.706,A -85,B 0,C 180,E1 -12310.112,E2 -12310.112} C_VEL
LIN {X 0,Y 381.167,Z 369.229,A -85,B 0,C 180,E1 -12310.765,E2 -12310.765} C_VEL
LIN {X 0,Y 379.784,Z 449.218,A -85,B 0,C 180,E1 -12312.469,E2 -12312.469} C_VEL
LIN {X 0,Y 379.401,Z 459.044,A -85,B 0,C 180,E1 -12312.798,E2 -12312.798} C_VEL
LIN {X 0,Y 378.962,Z 468.351,A -85,B 0,C 180,E1 -12313.229,E2 -12313.229} C_VEL
LIN {X 0,Y 378.435,Z 478.262,A -85,B 0,C 180,E1 -12313.829,E2 -12313.829} C_VEL
LIN {X 0,Y 377.785,Z 488.632,A -85,B 0,C 180,E1 -12314.631,E2 -12314.631} C_VEL
LIN {X 0,Y 377.251,Z 497.149,A -85,B 0,C 180,E1 -12315.438,E2 -12315.438} C_VEL
LIN {X 0,Y 376.695,Z 505.461,A -85,B 0,C 180,E1 -12316.38,E2 -12316.38} C_VEL
LIN {X 0,Y 376.059,Z 514.298,A -85,B 0,C 180,E1 -12317.593,E2 -12317.593} C_VEL
LIN {X 0,Y 375.613,Z 520.94,A -85,B 0,C 180,E1 -12318.673,E2 -12318.673} C_VEL
LIN {X 0,Y 375.198,Z 527.871,A -85,B 0,C 180,E1 -12320.025,E2 -12320.025} C_VEL
LIN {X 0,Y 374.929,Z 533.619,A -85,B 0,C 180,E1 -12321.379,E2 -12321.379} C_VEL
LIN {X 0,Y 374.722,Z 539.136,A -85,B 0,C 180,E1 -12323.001,E2 -12323.001} C_VEL
LIN {X 0,Y 374.611,Z 543.399,A -85,B 0,C 180,E1 -12324.62,E2 -12324.62} C_VEL
LIN {X 0,Y 374.611,Z 545.697,A -85,B 0,C 180,E1 -12325.699,E2 -12325.699} C_VEL
LIN {X 0,Y 374.707,Z 548.616,A -85,B 0,C 180,E1 -12327.853,E2 -12327.853} C_VEL
LIN {X 0,Y 374.66,Z 549.527,A -85,B 0,C 180,E1 -12328.927,E2 -12328.927} C_VEL
LIN {X 0,Y 374.649,Z 549.789,A -85,B 0,C 180,E1 -12331.077,E2 -12331.077} C_VEL
LIN {X 0,Y 374.625,Z 549.385,A -85,B 0,C 180,E1 -12332.152,E2 -12332.152} C_VEL
LIN {X 0,Y 374.576,Z 547.058,A -85,B 0,C 180,E1 -12334.306,E2 -12334.306} C_VEL
LIN {X 0,Y 374.565,Z 545.322,A -85,B 0,C 180,E1 -12335.385,E2 -12335.385} C_VEL
LIN {X 0,Y 374.717,Z 541.753,A -85,B 0,C 180,E1 -12337.004,E2 -12337.004} C_VEL
LIN {X 0,Y 374.936,Z 537.044,A -85,B 0,C 180,E1 -12338.626,E2 -12338.626} C_VEL
LIN {X 0,Y 375.358,Z 531.03,A -85,B 0,C 180,E1 -12340.247,E2 -12340.247} C_VEL
LIN {X 0,Y 376.009,Z 523.457,A -85,B 0,C 180,E1 -12341.866,E2 -12341.866} C_VEL
LIN {X 0,Y 376.731,Z 515.762,A -85,B 0,C 180,E1 -12343.211,E2 -12343.211} C_VEL
LIN {X 0,Y 377.399,Z 508.505,A -85,B 0,C 180,E1 -12344.281,E2 -12344.281} C_VEL
LIN {X 0,Y 378.238,Z 499.81,A -85,B 0,C 180,E1 -12345.354,E2 -12345.354} C_VEL
LIN {X 0,Y 379.093,Z 490.725,A -85,B 0,C 180,E1 -12346.285,E2 -12346.285} C_VEL
LIN {X 0,Y 379.962,Z 481.268,A -85,B 0,C 180,E1 -12347.076,E2 -12347.076} C_VEL
LIN {X 0,Y 380.791,Z 470.328,A -85,B 0,C 180,E1 -12347.8,E2 -12347.8} C_VEL
LIN {X 0,Y 381.423,Z 459.94,A -85,B 0,C 180,E1 -12348.324,E2 -12348.324} C_VEL
LIN {X 0,Y 381.952,Z 450.236,A -85,B 0,C 180,E1 -12348.68,E2 -12348.68} C_VEL
LIN {X 0,Y 382.54,Z 430.611,A -85,B 0,C 180,E1 -12349.137,E2 -12349.137} C_VEL
LIN {X 0,Y 383.81,Z 368.131,A -85,B 0,C 180,E1 -12350.53,E2 -12350.53} C_VEL
LIN {X 0,Y 381.243,Z 349.619,A -85,B 0,C 180,E1 -12351.177,E2 -12351.177} C_VEL
LIN {X 0,Y 380.147,Z 343.424,A -85,B 0,C 180,E1 -12351.427,E2 -12351.427} C_VEL
LIN {X 0,Y 382.212,Z 320.058,A -85,B 0,C 180,E1 -12355.426,E2 -12355.426} C_VEL
LIN {X 0,Y 381.69,Z 315.897,A -85,B 0,C 180,E1 -12356.225,E2 -12356.225} C_VEL
LIN {X 0,Y 379.174,Z 304.856,A -85,B 0,C 180,E1 -12358.507,E2 -12358.507} C_VEL
LIN {X 0,Y 376.533,Z 295.687,A -85,B 0,C 180,E1 -12360.538,E2 -12360.538} C_VEL
LIN {X 0,Y 375.951,Z 293.66,A -85,B 0,C 180,E1 -12361.014,E2 -12361.014} C_VEL
LIN {X 0,Y 375.972,Z 293.654,A -85,B 0,C 180,E1 -12364.667,E2 -12364.667} C_VEL
LIN {X 0,Y 375.964,Z 293.656,A -85,B 0,C 180,E1 -12368.269,E2 -12368.269} C_VEL
LIN {X 0,Y 375.924,Z 293.661,A -85,B 0,C 180,E1 -12371.6,E2 -12371.6} C_VEL
LIN {X 0,Y 375.915,Z 293.66,A -85,B 0,C 180,E1 -12375.268,E2 -12375.268} C_VEL
LIN {X 0,Y 375.961,Z 293.653,A -85,B 0,C 180,E1 -12379.136,E2 -12379.136} C_VEL
LIN {X 0,Y 375.951,Z 293.653,A -85,B 0,C 180,E1 -12381.911,E2 -12381.911} C_VEL
LIN {X 0,Y 375.963,Z 293.645,A -85,B 0,C 180,E1 -12385.332,E2 -12385.332} C_VEL
LIN {X 0,Y 375.94,Z 293.652,A -85,B 0,C 180,E1 -12388.437,E2 -12388.437} C_VEL
LIN {X 0,Y 375.977,Z 293.645,A -85,B 0,C 180,E1 -12392.14,E2 -12392.14} C_VEL
LIN {X 0,Y 375.986,Z 293.648,A -85,B 0,C 180,E1 -12394.538,E2 -12394.538} C_VEL
LIN {X 0,Y 375.973,Z 293.653,A -85,B 0,C 180,E1 -12398.047,E2 -12398.047} C_VEL
LIN {X 0,Y 376.008,Z 293.648,A -85,B 0,C 180,E1 -12401.474,E2 -12401.474} C_VEL
LIN {X 0,Y 376.035,Z 293.645,A -85,B 0,C 180,E1 -12404.832,E2 -12404.832} C_VEL
LIN {X 0,Y 376.034,Z 293.645,A -85,B 0,C 180,E1 -12408.137,E2 -12408.137} C_VEL
LIN {X 0,Y 376.194,Z 293.631,A -85,B 0,C 180,E1 -12411.922,E2 -12411.922} C_VEL
LIN {X 0,Y 376.197,Z 293.638,A -85,B 0,C 180,E1 -12413.295,E2 -12413.295} C_VEL
LIN {X 0,Y 380.469,Z 309.115,A -85,B 0,C 180,E1 -12416.533,E2 -12416.533} C_VEL
LIN {X 0,Y 379.748,Z 323.203,A -85,B 0,C 180,E1 -12418.94,E2 -12418.94} C_VEL
LIN {X 0,Y 379.096,Z 338.407,A -85,B 0,C 180,E1 -12421.502,E2 -12421.502} C_VEL
LIN {X 0,Y 382.595,Z 356.813,A -85,B 0,C 180,E1 -12422.288,E2 -12422.288} C_VEL
LIN {X 0,Y 383.529,Z 362.961,A -85,B 0,C 180,E1 -12422.531,E2 -12422.531} C_VEL
LIN {X 0,Y 381.556,Z 424.794,A -85,B 0,C 180,E1 -12424.135,E2 -12424.135} C_VEL
LIN {X 0,Y 381.049,Z 436.461,A -85,B 0,C 180,E1 -12424.61,E2 -12424.61} C_VEL
LIN {X 0,Y 380.369,Z 447.902,A -85,B 0,C 180,E1 -12425.301,E2 -12425.301} C_VEL
LIN {X 0,Y 379.74,Z 457.908,A -85,B 0,C 180,E1 -12426.109,E2 -12426.109} C_VEL
LIN {X 0,Y 379.13,Z 464.84,A -85,B 0,C 180,E1 -12426.787,E2 -12426.787} C_VEL
LIN {X 0,Y 378.402,Z 472.882,A -85,B 0,C 180,E1 -12427.739,E2 -12427.739} C_VEL
LIN {X 0,Y 377.673,Z 480.318,A -85,B 0,C 180,E1 -12428.81,E2 -12428.81} C_VEL
LIN {X 0,Y 377.035,Z 486.719,A -85,B 0,C 180,E1 -12429.929,E2 -12429.929} C_VEL
LIN {X 0,Y 376.405,Z 493.164,A -85,B 0,C 180,E1 -12431.307,E2 -12431.307} C_VEL
LIN {X 0,Y 375.725,Z 499.121,A -85,B 0,C 180,E1 -12432.972,E2 -12432.972} C_VEL
LIN {X 0,Y 375.42,Z 502.227,A -85,B 0,C 180,E1 -12434.086,E2 -12434.086} C_VEL
LIN {X 0,Y 375.162,Z 504.641,A -85,B 0,C 180,E1 -12435.205,E2 -12435.205} C_VEL
LIN {X 0,Y 374.818,Z 507.233,A -85,B 0,C 180,E1 -12437.018,E2 -12437.018} C_VEL
LIN {X 0,Y 374.594,Z 508.271,A -85,B 0,C 180,E1 -12438.6,E2 -12438.6} C_VEL
LIN {X 0,Y 374.545,Z 508.169,A -85,B 0,C 180,E1 -12440.257,E2 -12440.257} C_VEL
LIN {X 0,Y 374.516,Z 507.89,A -85,B 0,C 180,E1 -12440.889,E2 -12440.889} C_VEL
LIN {X 0,Y 374.571,Z 506.741,A -85,B 0,C 180,E1 -12442.041,E2 -12442.041} C_VEL
LIN {X 0,Y 374.787,Z 503.905,A -85,B 0,C 180,E1 -12443.776,E2 -12443.776} C_VEL
LIN {X 0,Y 374.938,Z 501.168,A -85,B 0,C 180,E1 -12444.946,E2 -12444.946} C_VEL
LIN {X 0,Y 375.137,Z 497.139,A -85,B 0,C 180,E1 -12446.272,E2 -12446.272} C_VEL
LIN {X 0,Y 375.447,Z 491.994,A -85,B 0,C 180,E1 -12447.601,E2 -12447.601} C_VEL
LIN {X 0,Y 375.855,Z 485.69,A -85,B 0,C 180,E1 -12448.903,E2 -12448.903} C_VEL
LIN {X 0,Y 376.248,Z 479.378,A -85,B 0,C 180,E1 -12449.979,E2 -12449.979} C_VEL
LIN {X 0,Y 376.624,Z 473.191,A -85,B 0,C 180,E1 -12450.87,E2 -12450.87} C_VEL
LIN {X 0,Y 377.105,Z 465.733,A -85,B 0,C 180,E1 -12451.769,E2 -12451.769} C_VEL
LIN {X 0,Y 377.612,Z 456.626,A -85,B 0,C 180,E1 -12452.667,E2 -12452.667} C_VEL
LIN {X 0,Y 377.973,Z 448.93,A -85,B 0,C 180,E1 -12453.286,E2 -12453.286} C_VEL
LIN {X 0,Y 378.363,Z 439.956,A -85,B 0,C 180,E1 -12453.866,E2 -12453.866} C_VEL
LIN {X 0,Y 378.714,Z 429.558,A -85,B 0,C 180,E1 -12454.372,E2 -12454.372} C_VEL
LIN {X 0,Y 379.01,Z 417.401,A -85,B 0,C 180,E1 -12454.765,E2 -12454.765} C_VEL
LIN {X 0,Y 380.073,Z 361.395,A -85,B 0,C 180,E1 -12456.064,E2 -12456.064} C_VEL
LIN {X 0,Y 376.991,Z 339.49,A -85,B 0,C 180,E1 -12456.719,E2 -12456.719} C_VEL
LIN {X 0,Y 377.841,Z 325.068,A -85,B 0,C 180,E1 -12459.92,E2 -12459.92} C_VEL
LIN {X 0,Y 378.739,Z 311.466,A -85,B 0,C 180,E1 -12462.996,E2 -12462.996} C_VEL
LIN {X 0,Y 378.852,Z 308.577,A -85,B 0,C 180,E1 -12463.66,E2 -12463.66} C_VEL
LIN {X 0,Y 376.507,Z 296.256,A -85,B 0,C 180,E1 -12466.719,E2 -12466.719} C_VEL
LIN {X 0,Y 375.972,Z 293.653,A -85,B 0,C 180,E1 -12467.377,E2 -12467.377} C_VEL
LIN {X 0,Y 375.931,Z 293.654,A -85,B 0,C 180,E1 -12470.535,E2 -12470.535} C_VEL
LIN {X 0,Y 375.954,Z 293.656,A -85,B 0,C 180,E1 -12473.499,E2 -12473.499} C_VEL
LIN {X 0,Y 375.956,Z 293.656,A -85,B 0,C 180,E1 -12475.889,E2 -12475.889} C_VEL
LIN {X 0,Y 375.961,Z 293.653,A -85,B 0,C 180,E1 -12479.688,E2 -12479.688} C_VEL
LIN {X 0,Y 375.919,Z 293.662,A -85,B 0,C 180,E1 -12482.136,E2 -12482.136} C_VEL
LIN {X 0,Y 375.938,Z 293.656,A -85,B 0,C 180,E1 -12484.534,E2 -12484.534} C_VEL
LIN {X 0,Y 375.973,Z 293.65,A -85,B 0,C 180,E1 -12486.887,E2 -12486.887} C_VEL
LIN {X 0,Y 375.989,Z 293.65,A -85,B 0,C 180,E1 -12490.339,E2 -12490.339} C_VEL
LIN {X 0,Y 376.027,Z 293.641,A -85,B 0,C 180,E1 -12493.718,E2 -12493.718} C_VEL
LIN {X 0,Y 376.109,Z 293.638,A -85,B 0,C 180,E1 -12497.041,E2 -12497.041} C_VEL
LIN {X 0,Y 376.114,Z 293.63,A -85,B 0,C 180,E1 -12500.317,E2 -12500.317} C_VEL
LIN {X 0,Y 376.198,Z 293.624,A -85,B 0,C 180,E1 -12503.563,E2 -12503.563} C_VEL
LIN {X 0,Y 376.336,Z 293.607,A -85,B 0,C 180,E1 -12507.858,E2 -12507.858} C_VEL
LIN {X 0,Y 376.335,Z 293.606,A -85,B 0,C 180,E1 -12512.138,E2 -12512.138} C_VEL
LIN {X 0,Y 376.195,Z 293.623,A -85,B 0,C 180,E1 -12516.433,E2 -12516.433} C_VEL
LIN {X 0,Y 376.11,Z 293.632,A -85,B 0,C 180,E1 -12519.679,E2 -12519.679} C_VEL
LIN {X 0,Y 376.045,Z 293.639,A -85,B 0,C 180,E1 -12521.957,E2 -12521.957} C_VEL
LIN {X 0,Y 375.385,Z 293.724,A -85,B 0,C 180,E1 -12522.85,E2 -12522.85} C_VEL
LIN {X 0,Y 372.533,Z 294.084,A -85,B 0,C 180,E1 -12524.303,E2 -12524.303} C_VEL
LIN {X 0,Y 370.105,Z 294.391,A -85,B 0,C 180,E1 -12525.477,E2 -12525.477} C_VEL
LIN {X 0,Y 369.053,Z 294.518,A -85,B 0,C 180,E1 -12526.386,E2 -12526.386} C_VEL
LIN {X 0,Y 368.962,Z 294.526,A -85,B 0,C 180,E1 -12526.694,E2 -12526.694} C_VEL
LIN {X 0,Y 368.93,Z 294.525,A -85,B 0,C 180,E1 -12530.049,E2 -12530.049} C_VEL
LIN {X 0,Y 368.915,Z 294.527,A -85,B 0,C 180,E1 -12533.875,E2 -12533.875} C_VEL
LIN {X 0,Y 368.857,Z 294.54,A -85,B 0,C 180,E1 -12537.206,E2 -12537.206} C_VEL
LIN {X 0,Y 368.882,Z 294.535,A -85,B 0,C 180,E1 -12539.687,E2 -12539.687} C_VEL
LIN {X 0,Y 368.881,Z 294.532,A -85,B 0,C 180,E1 -12543.038,E2 -12543.038} C_VEL
LIN {X 0,Y 368.898,Z 294.532,A -85,B 0,C 180,E1 -12546.192,E2 -12546.192} C_VEL
LIN {X 0,Y 368.876,Z 294.531,A -85,B 0,C 180,E1 -12548.949,E2 -12548.949} C_VEL
LIN {X 0,Y 368.851,Z 294.54,A -85,B 0,C 180,E1 -12552.003,E2 -12552.003} C_VEL
LIN {X 0,Y 368.851,Z 294.535,A -85,B 0,C 180,E1 -12555.171,E2 -12555.171} C_VEL
LIN {X 0,Y 368.852,Z 294.538,A -85,B 0,C 180,E1 -12558.173,E2 -12558.173} C_VEL
LIN {X 0,Y 368.874,Z 294.532,A -85,B 0,C 180,E1 -12561.356,E2 -12561.356} C_VEL
LIN {X 0,Y 368.894,Z 294.534,A -85,B 0,C 180,E1 -12565.141,E2 -12565.141} C_VEL
LIN {X 0,Y 368.892,Z 294.536,A -85,B 0,C 180,E1 -12569.042,E2 -12569.042} C_VEL
LIN {X 0,Y 368.94,Z 294.527,A -85,B 0,C 180,E1 -12571.56,E2 -12571.56} C_VEL
LIN {X 0,Y 368.957,Z 294.523,A -85,B 0,C 180,E1 -12574.016,E2 -12574.016} C_VEL
LIN {X 0,Y 368.876,Z 294.539,A -85,B 0,C 180,E1 -12577.601,E2 -12577.601} C_VEL
LIN {X 0,Y 368.886,Z 294.531,A -85,B 0,C 180,E1 -12581.101,E2 -12581.101} C_VEL
LIN {X 0,Y 368.948,Z 294.524,A -85,B 0,C 180,E1 -12584.532,E2 -12584.532} C_VEL
LIN {X 0,Y 368.961,Z 294.525,A -85,B 0,C 180,E1 -12587.905,E2 -12587.905} C_VEL
LIN {X 0,Y 369.116,Z 294.503,A -85,B 0,C 180,E1 -12591.868,E2 -12591.868} C_VEL
LIN {X 0,Y 369.092,Z 294.512,A -85,B 0,C 180,E1 -12594.536,E2 -12594.536} C_VEL
LIN {X 0,Y 369.27,Z 294.482,A -85,B 0,C 180,E1 -12597.818,E2 -12597.818} C_VEL
LIN {X 0,Y 369.404,Z 294.466,A -85,B 0,C 180,E1 -12599.999,E2 -12599.999} C_VEL
LIN {X 0,Y 369.266,Z 294.483,A -85,B 0,C 180,E1 -12602.181,E2 -12602.181} C_VEL
LIN {X 0,Y 369.149,Z 294.498,A -85,B 0,C 180,E1 -12606.559,E2 -12606.559} C_VEL
LIN {X 0,Y 369.016,Z 294.517,A -85,B 0,C 180,E1 -12609.869,E2 -12609.869} C_VEL
LIN {X 0,Y 368.987,Z 294.524,A -85,B 0,C 180,E1 -12613.773,E2 -12613.773} C_VEL
LIN {X 0,Y 368.954,Z 294.528,A -85,B 0,C 180,E1 -12617.77,E2 -12617.77} C_VEL
LIN {X 0,Y 368.864,Z 294.533,A -85,B 0,C 180,E1 -12621.223,E2 -12621.223} C_VEL
LIN {X 0,Y 368.911,Z 294.529,A -85,B 0,C 180,E1 -12624.778,E2 -12624.778} C_VEL
LIN {X 0,Y 368.917,Z 294.527,A -85,B 0,C 180,E1 -12627.206,E2 -12627.206} C_VEL
LIN {X 0,Y 368.869,Z 294.536,A -85,B 0,C 180,E1 -12630.991,E2 -12630.991} C_VEL
LIN {X 0,Y 368.896,Z 294.536,A -85,B 0,C 180,E1 -12634.857,E2 -12634.857} C_VEL
LIN {X 0,Y 368.865,Z 294.535,A -85,B 0,C 180,E1 -12638.643,E2 -12638.643} C_VEL
LIN {X 0,Y 368.843,Z 294.536,A -85,B 0,C 180,E1 -12642.012,E2 -12642.012} C_VEL
LIN {X 0,Y 368.846,Z 294.539,A -85,B 0,C 180,E1 -12645.179,E2 -12645.179} C_VEL
LIN {X 0,Y 368.852,Z 294.536,A -85,B 0,C 180,E1 -12648.181,E2 -12648.181} C_VEL
